(* PLC project AutomationML, AutomationML AutomationML AutomationML, author AutomationML *)
(* stored: creationDateTime 2017-02-14T12:09:57, companyURL AutomationML, productRelease AutomationML, language en-US, version AutomationML, organization AutomationML, modificationDateTime 2022-02-26T19:00:26 *)

PROGRAM Sequencing_Station_ActivityOnNodeNetwork
  VAR
    TA_030RB_300_takes_over_good : BOOL;
    TA_005RB_002_positions_workpiece1 : BOOL;
    TA_005RB_001_takes_over_workpiece1 : BOOL;
    TA_004CT_001_execute_trimming : BOOL;
    TA_003RB_002_positions_workpiece1 : BOOL;
    TA_001RB_001_takes_over_blank : BOOL;
    TA_001RB_002_positions_blank : BOOL;
    TA_030GST100_declamps_good : BOOL;
    TA_Execute_manufacturing_030RB_200 : BOOL;
    TA_Execute_manufacturing_030RB_100 : BOOL;
    TA_030GST100_clamps_goods : BOOL;
    TA_010RB_100_positions_workpiece1 : BOOL;
    TA_010RB_100_takes_over_workpiece1 : BOOL;
    TA_002DDP_001_execute_forming : BOOL;
    TA_003RB_001_takes_over_workpiece1 : BOOL;
    TA_006CMM_001_execute_cmm : BOOL;
    TA_007RB_001_takes_over_hinge_reinforcement : BOOL;
    TA_007RB_001_positions_hinge_reinforcement : BOOL;
    TA_030RB_300_positions_good : BOOL;
    TA_010UT_001_execute_inspection : BOOL;
  END_VAR

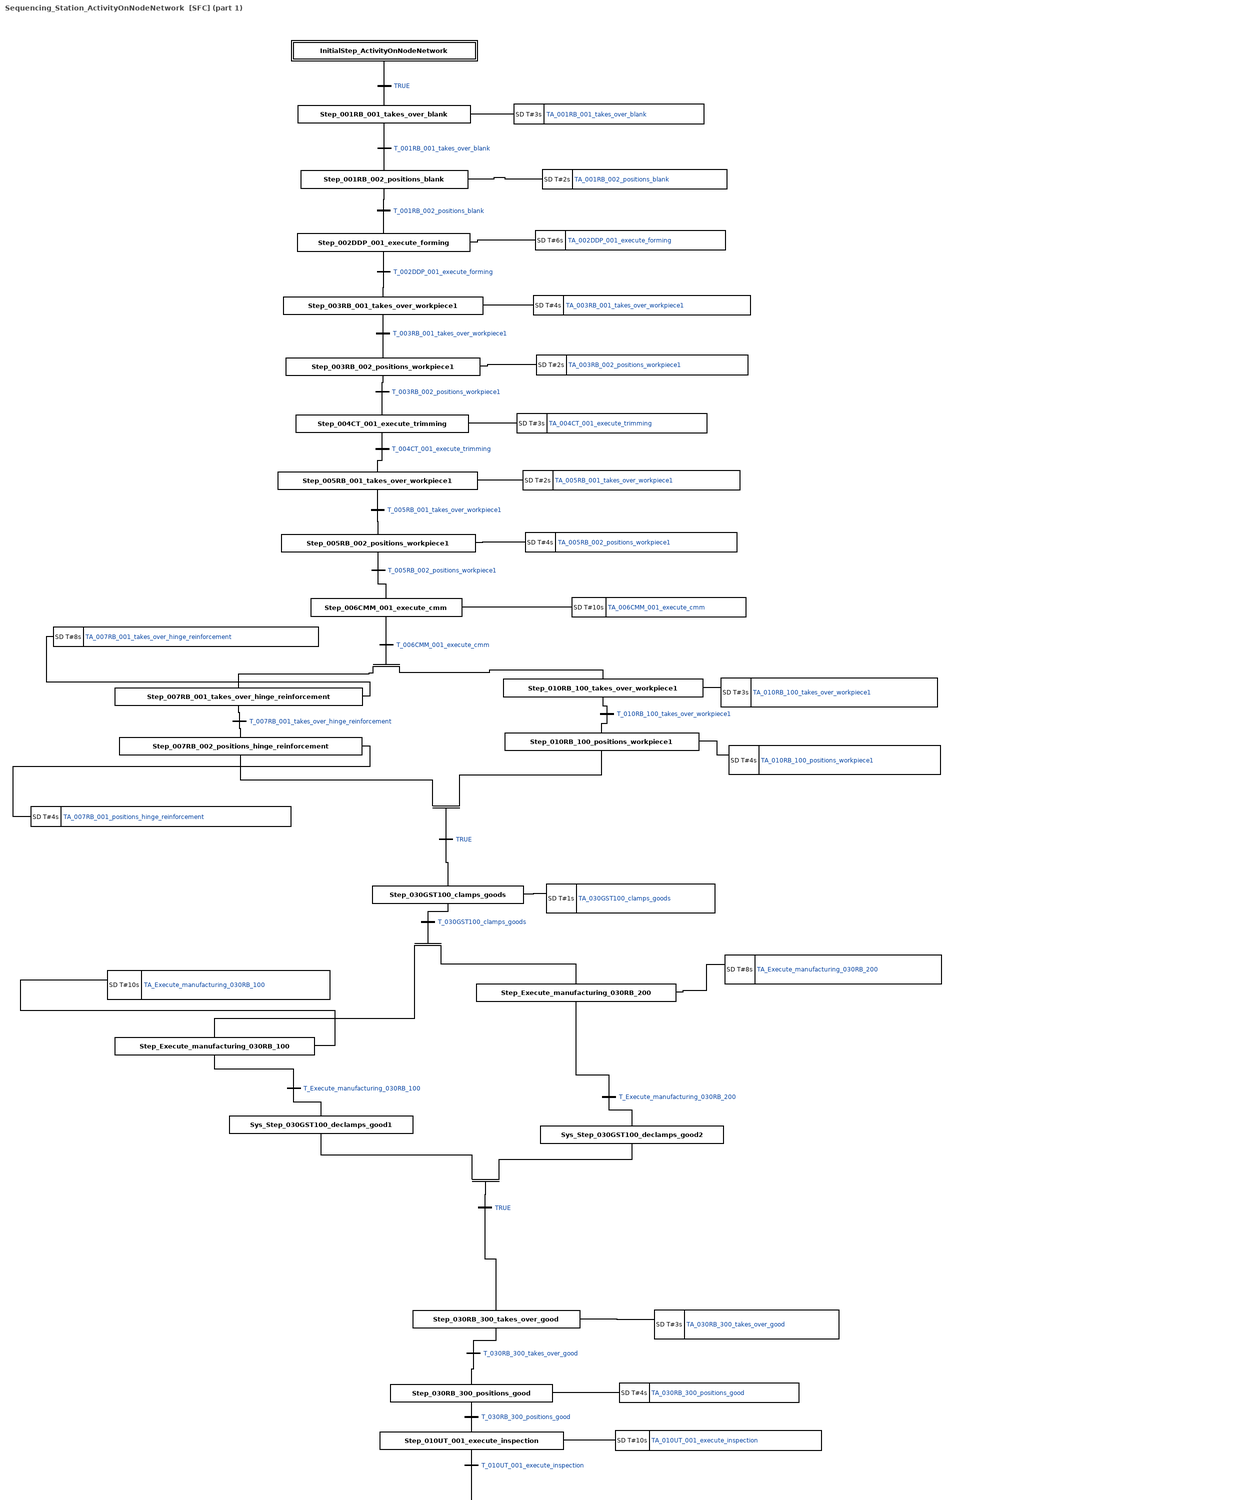
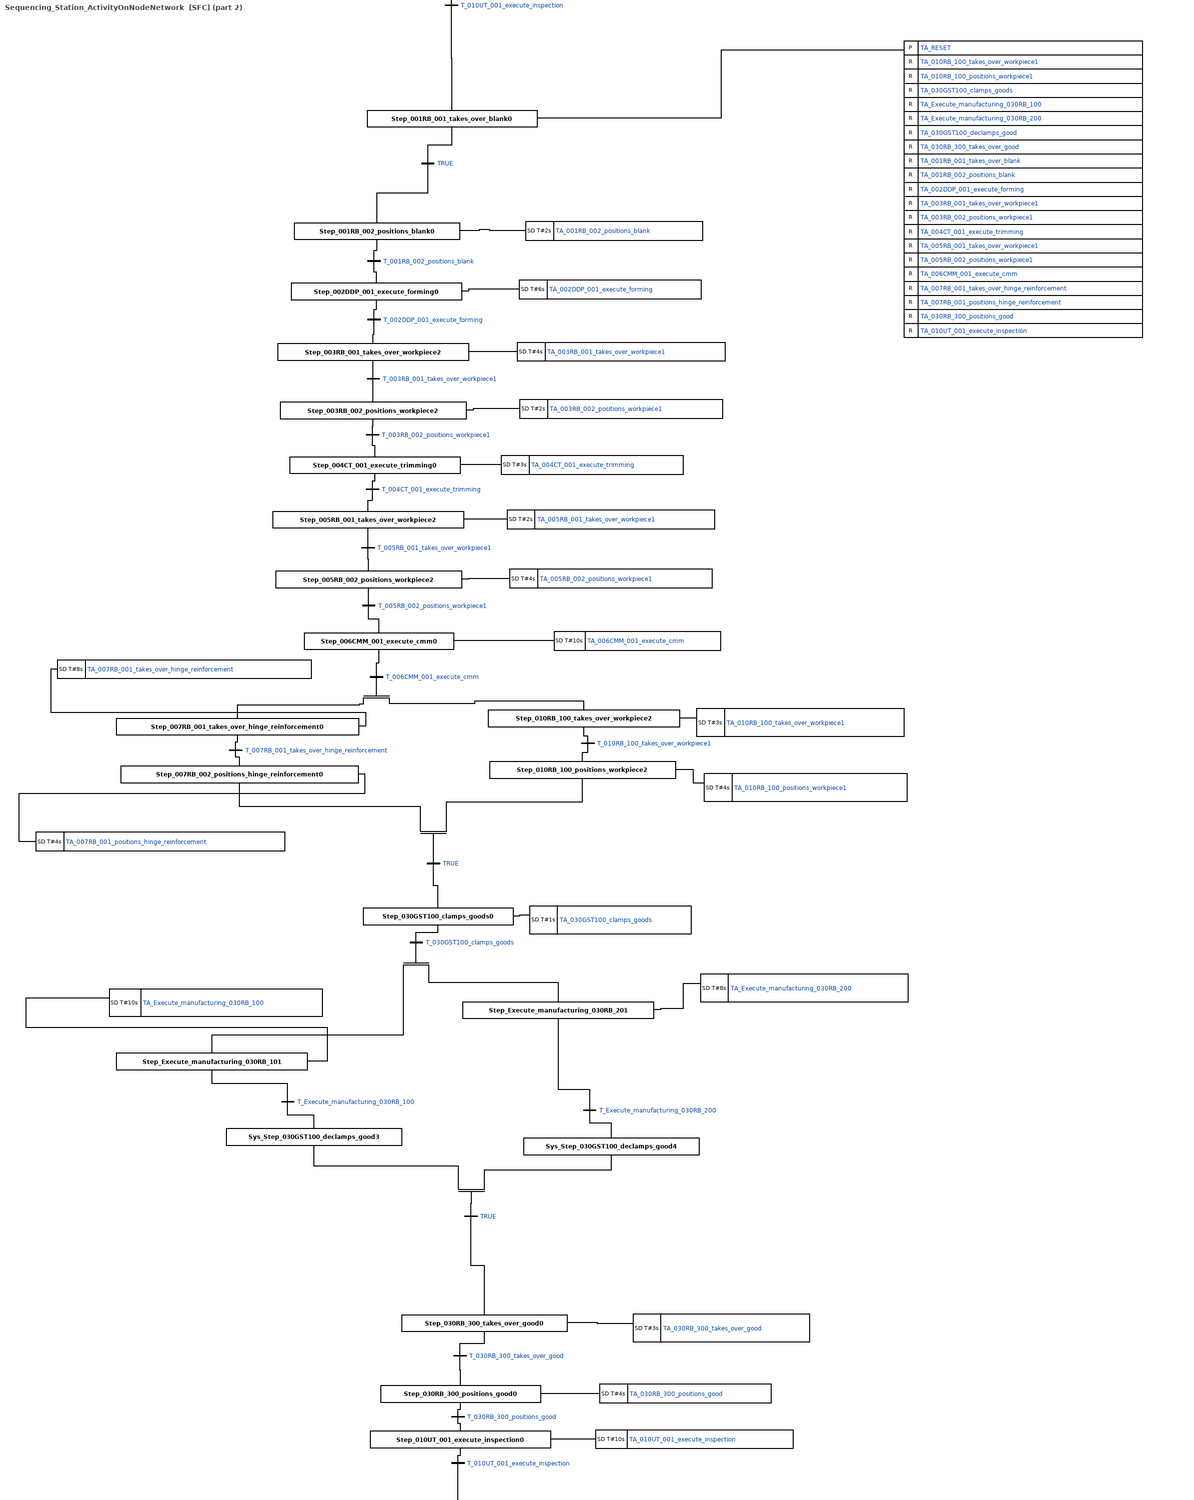
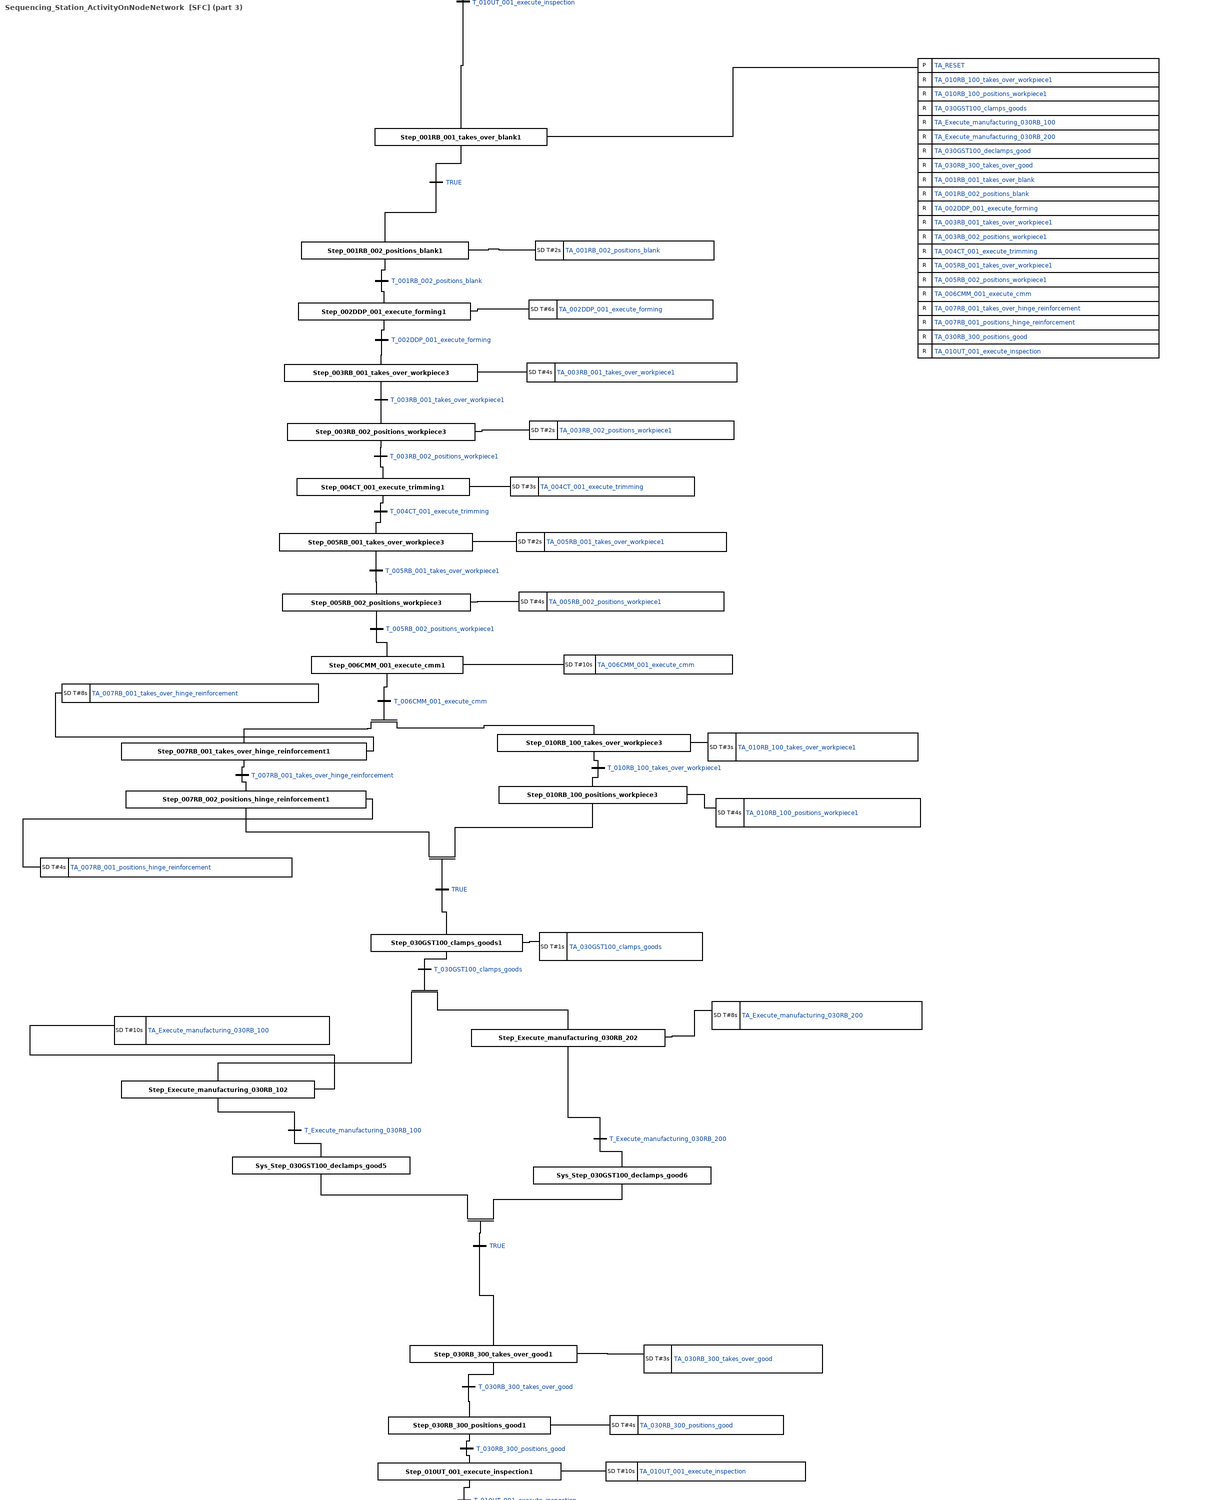
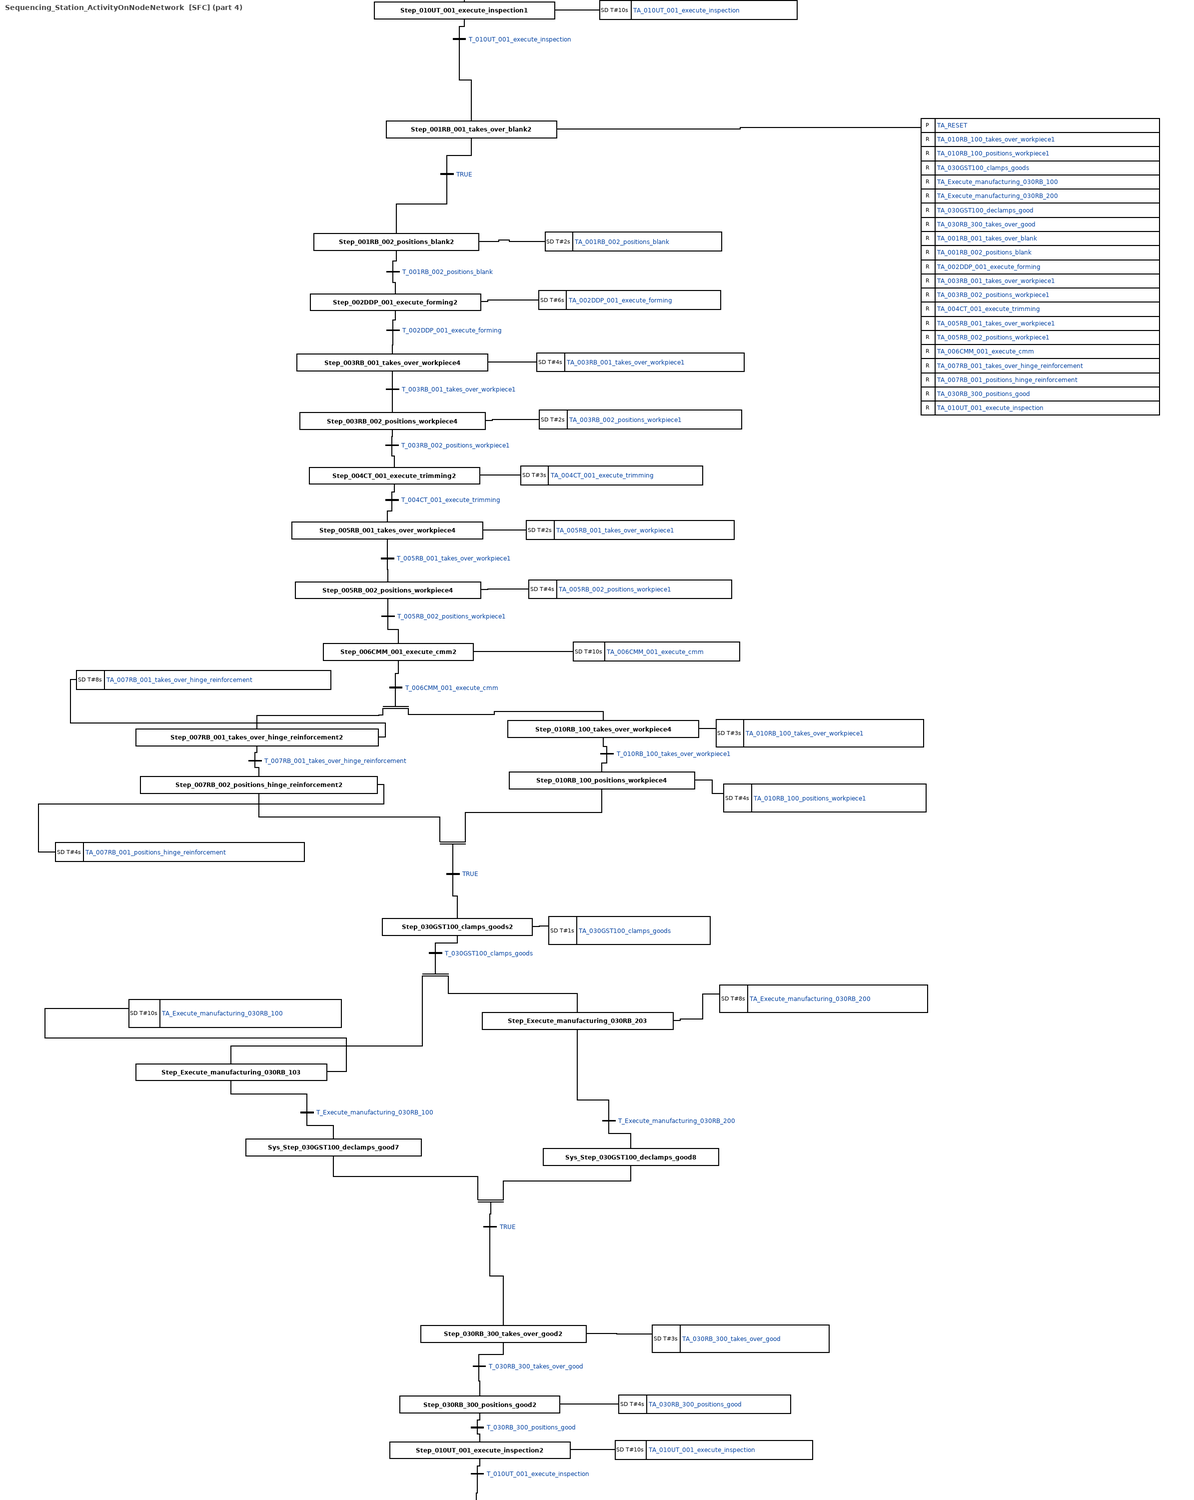
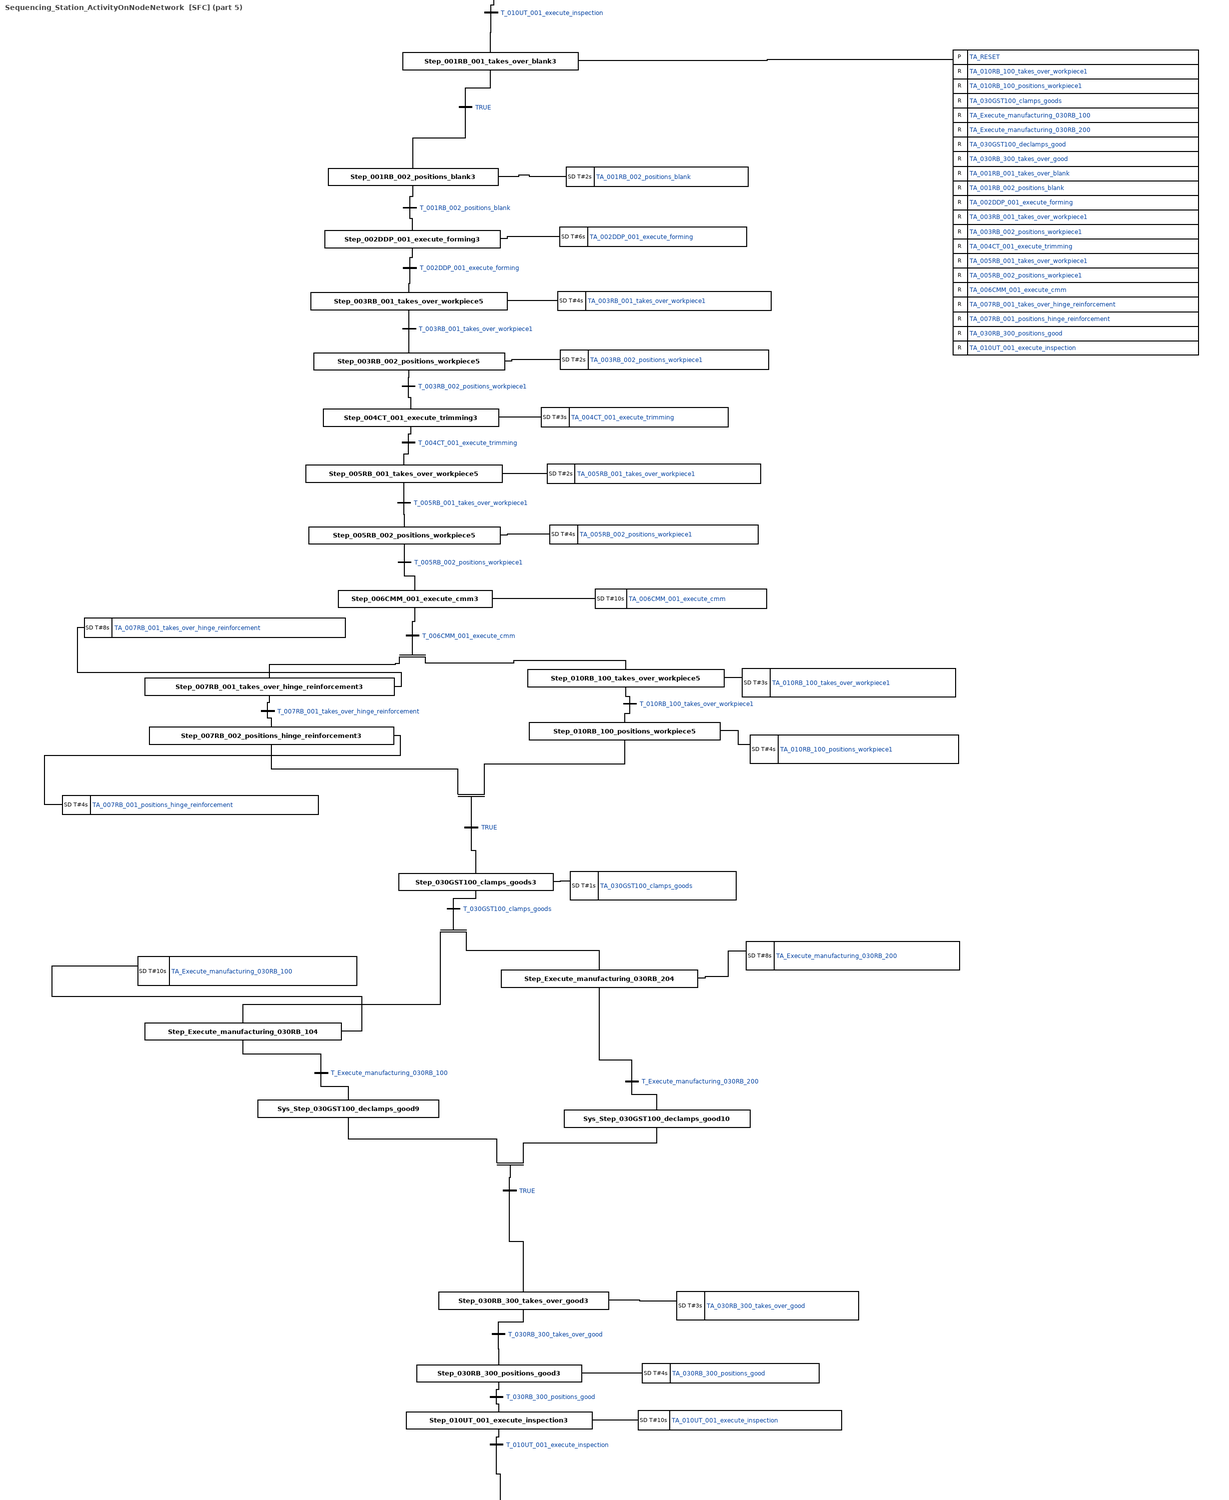
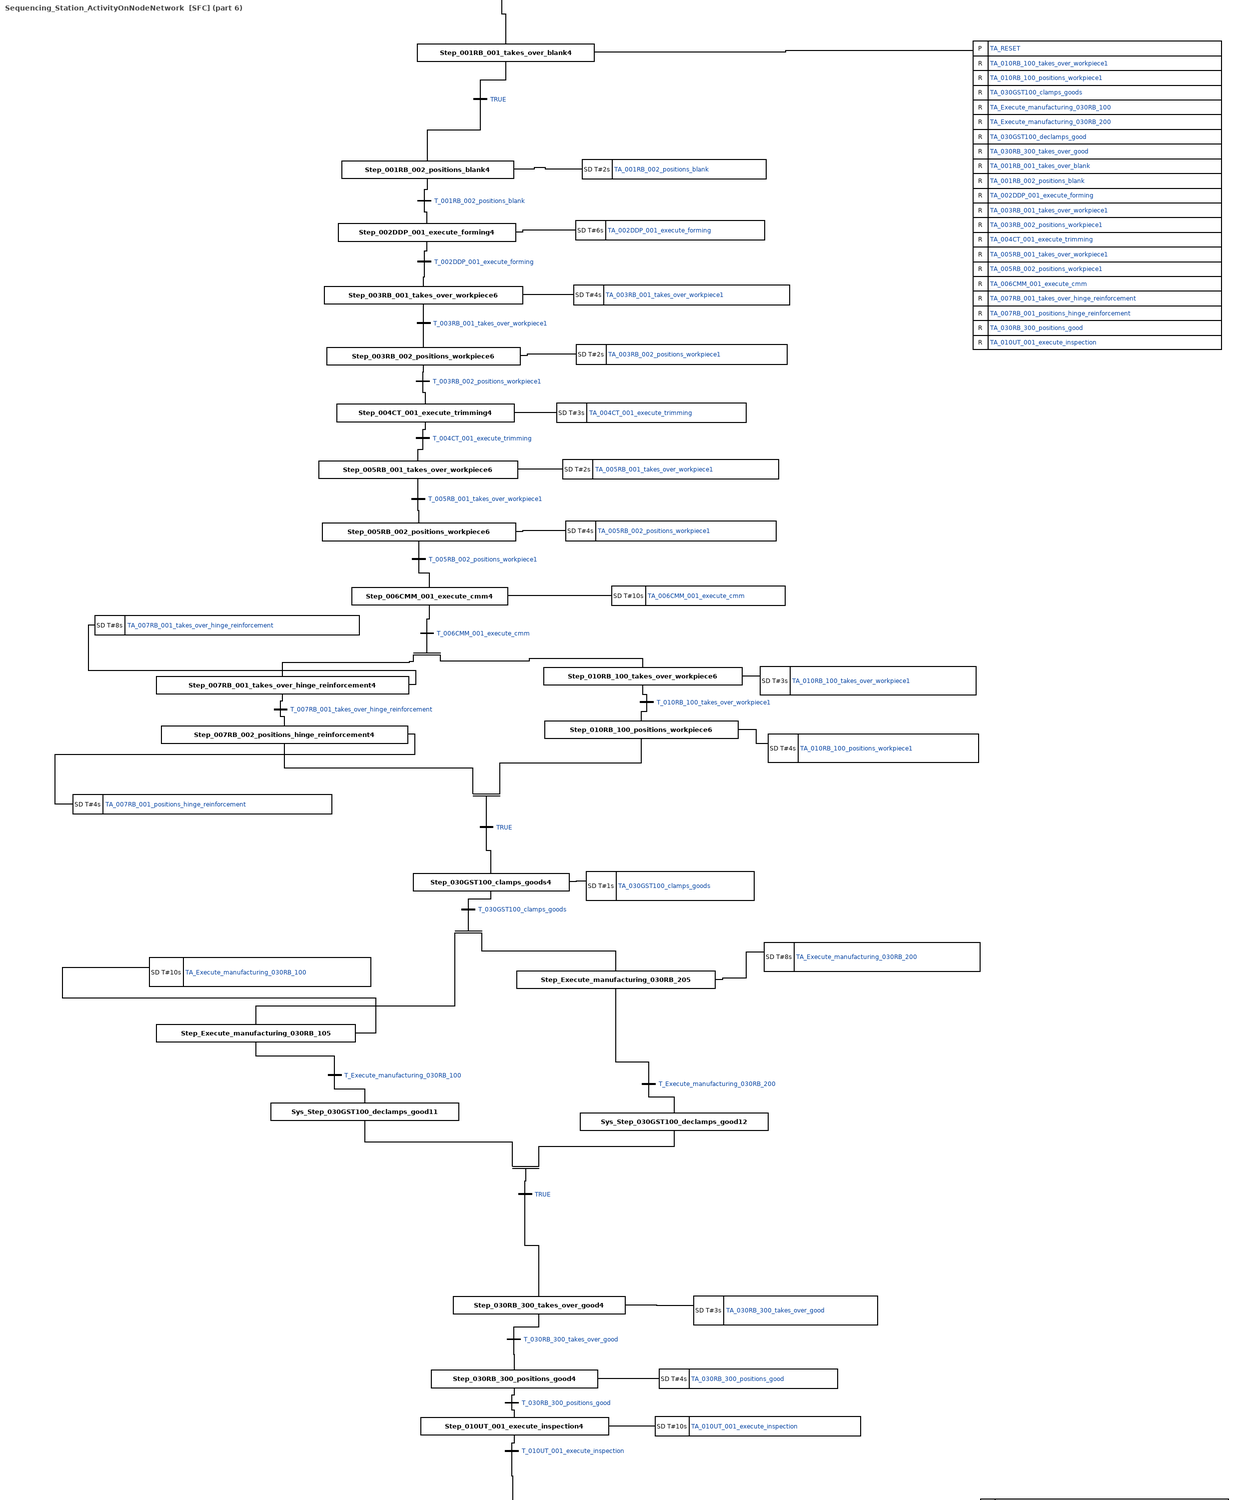
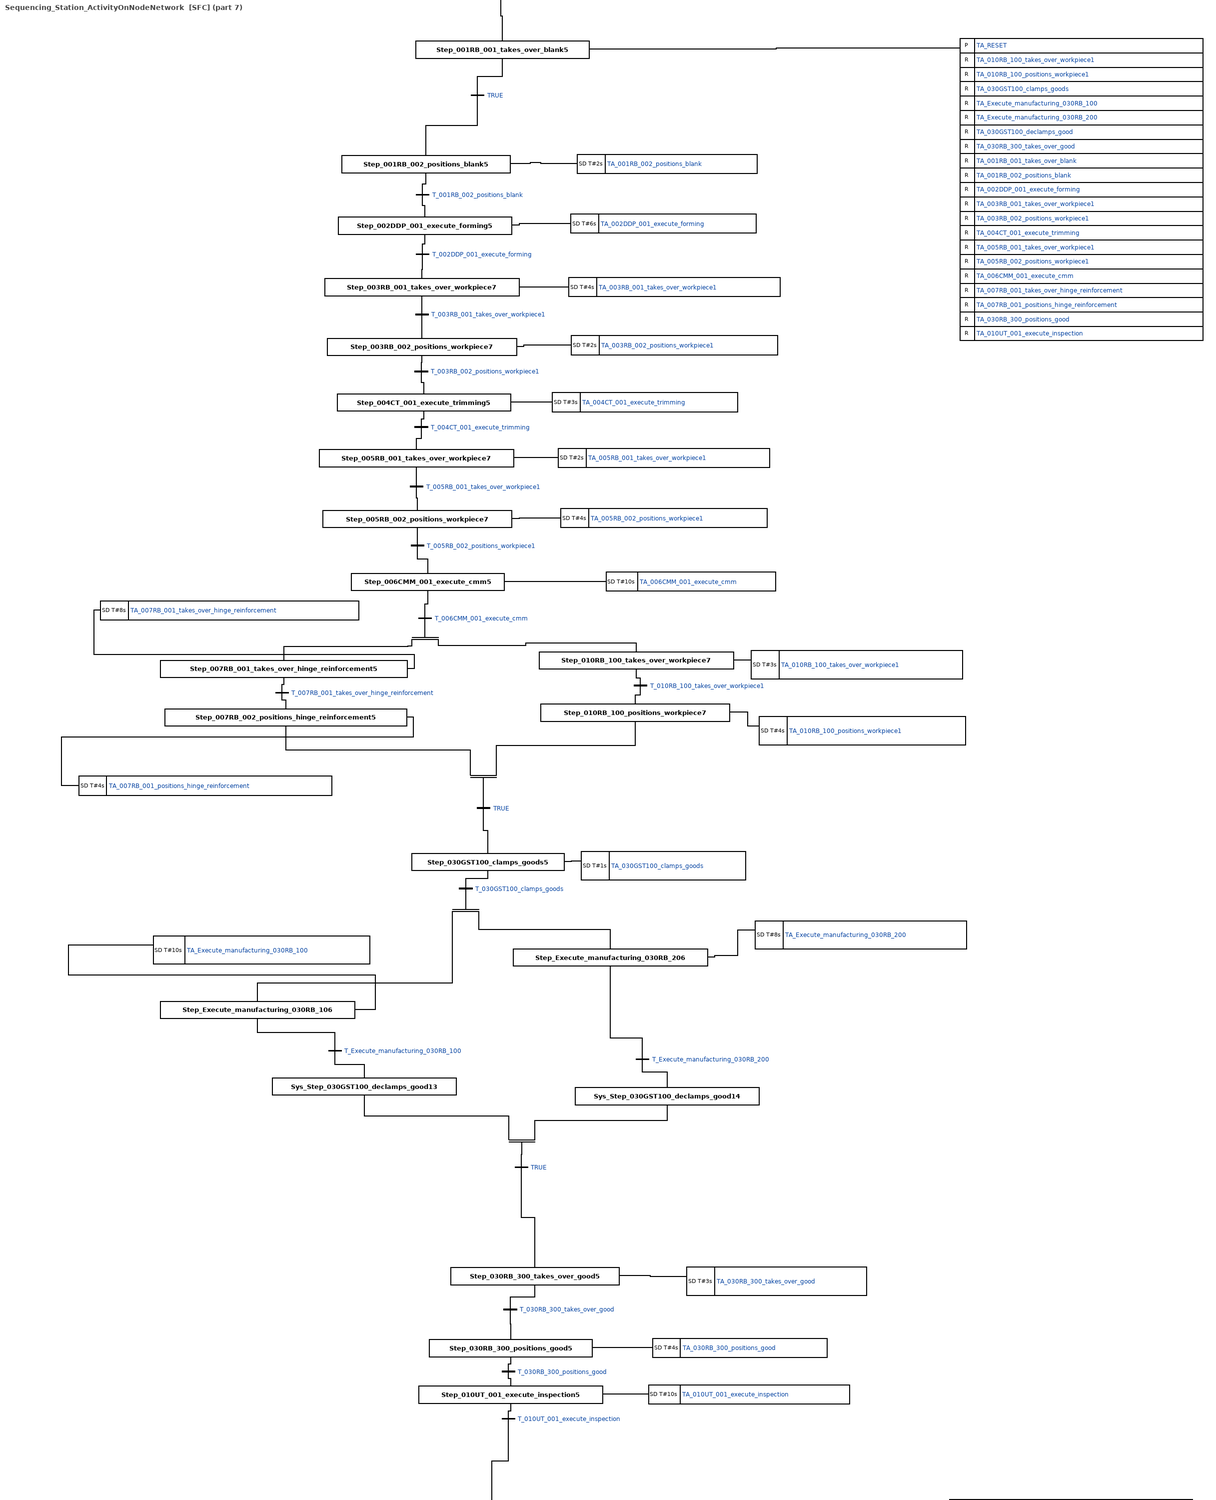
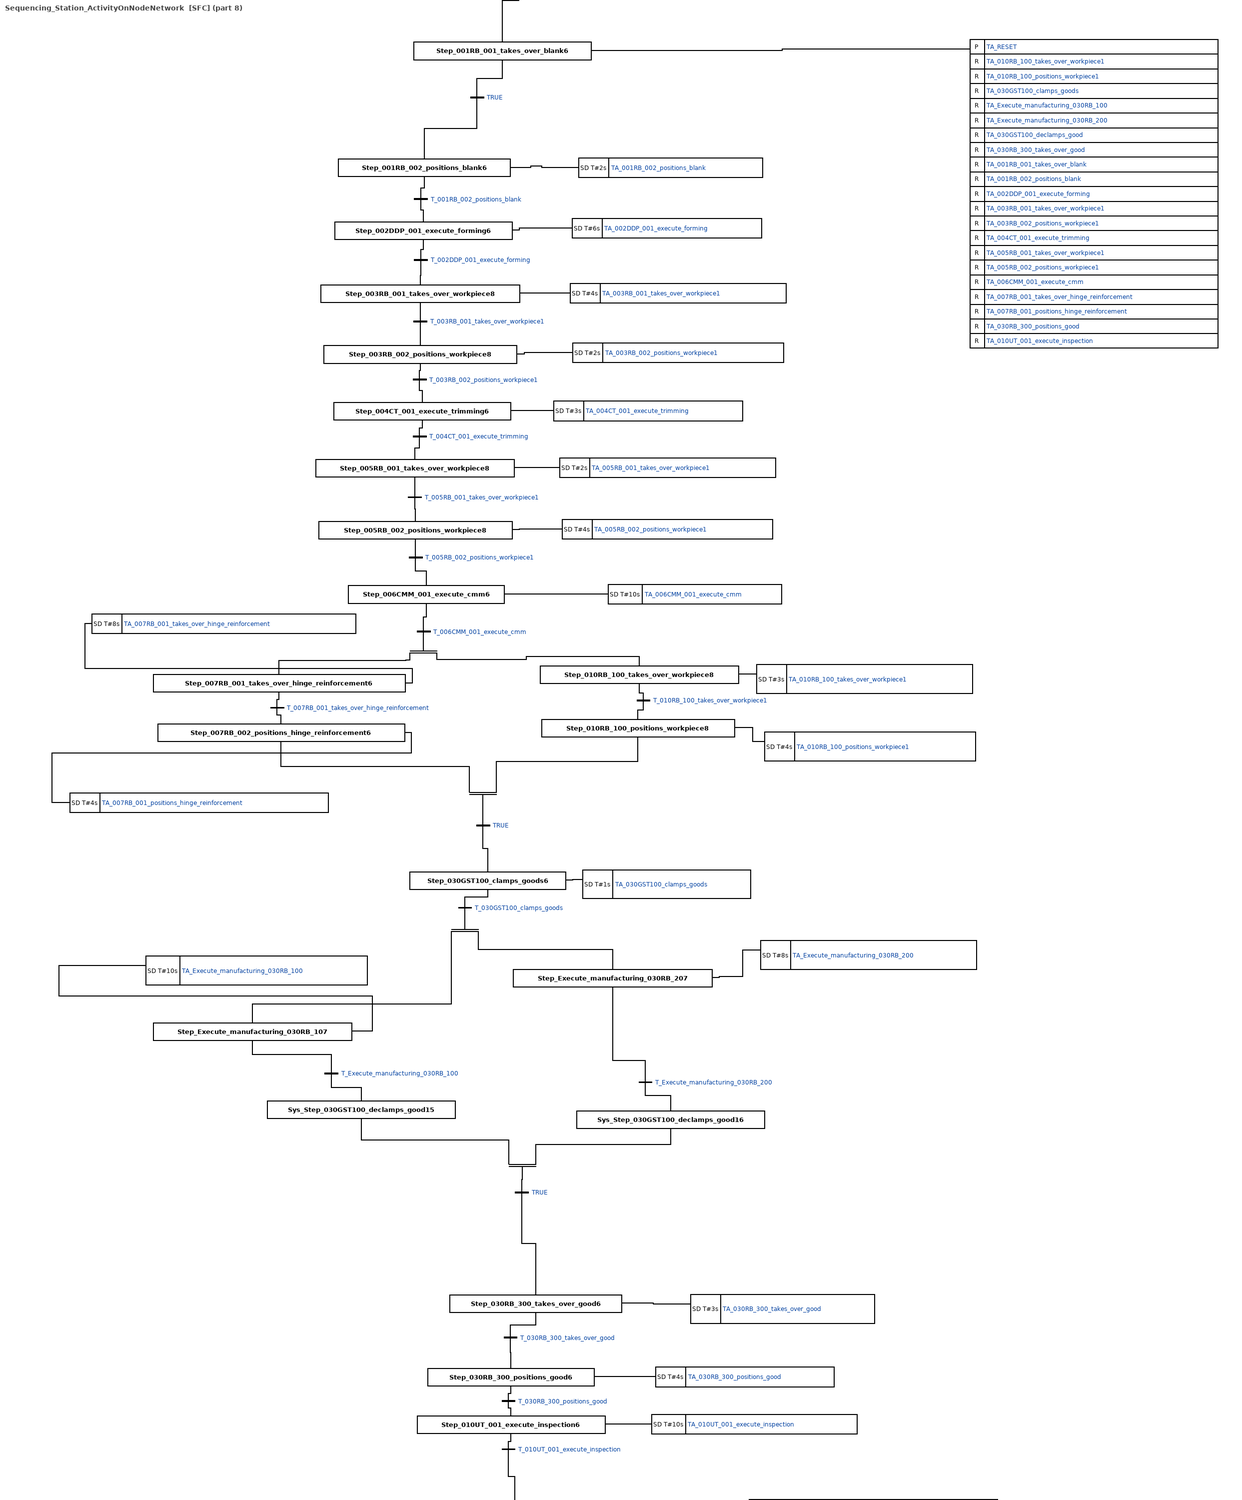
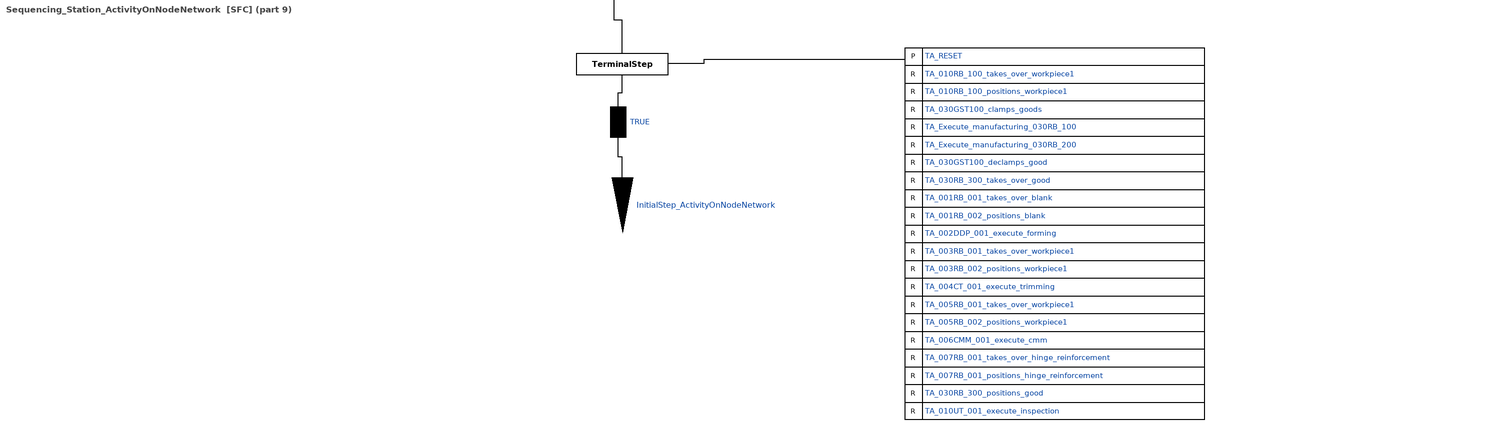
INITIAL_STEP InitialStep_ActivityOnNodeNetwork:
END_STEP
TRANSITION FROM InitialStep_ActivityOnNodeNetwork TO Step_001RB_001_takes_over_blank
  := TRUE;
END_TRANSITION
STEP Step_001RB_001_takes_over_blank:
  TA_001RB_001_takes_over_blank(SD, T#3s);
END_STEP
TRANSITION FROM Step_001RB_001_takes_over_blank TO Step_001RB_002_positions_blank  (* T_001RB_001_takes_over_blank *)
  := TA_001RB_001_takes_over_blank;
END_TRANSITION
STEP Step_001RB_002_positions_blank:
  TA_001RB_002_positions_blank(SD, T#2s);
END_STEP
TRANSITION FROM Step_001RB_002_positions_blank TO Step_002DDP_001_execute_forming  (* T_001RB_002_positions_blank *)
  := TA_001RB_002_positions_blank;
END_TRANSITION
STEP Step_002DDP_001_execute_forming:
  TA_002DDP_001_execute_forming(SD, T#6s);
END_STEP
TRANSITION FROM Step_002DDP_001_execute_forming TO Step_003RB_001_takes_over_workpiece1  (* T_002DDP_001_execute_forming *)
  := TA_002DDP_001_EXECUTE_FORMING;
END_TRANSITION
STEP Step_003RB_001_takes_over_workpiece1:
  TA_003RB_001_takes_over_workpiece1(SD, T#4s);
END_STEP
TRANSITION FROM Step_003RB_001_takes_over_workpiece1 TO Step_003RB_002_positions_workpiece1  (* T_003RB_001_takes_over_workpiece1 *)
  := TA_003RB_001_takes_over_workpiece1;
END_TRANSITION
STEP Step_003RB_002_positions_workpiece1:
  TA_003RB_002_positions_workpiece1(SD, T#2s);
END_STEP
TRANSITION FROM Step_003RB_002_positions_workpiece1 TO Step_004CT_001_execute_trimming  (* T_003RB_002_positions_workpiece1 *)
  := TA_003RB_002_positions_workpiece1;
END_TRANSITION
STEP Step_004CT_001_execute_trimming:
  TA_004CT_001_execute_trimming(SD, T#3s);
END_STEP
TRANSITION FROM Step_004CT_001_execute_trimming TO Step_005RB_001_takes_over_workpiece1  (* T_004CT_001_execute_trimming *)
  := TA_004CT_001_execute_trimming;
END_TRANSITION
STEP Step_005RB_001_takes_over_workpiece1:
  TA_005RB_001_takes_over_workpiece1(SD, T#2s);
END_STEP
TRANSITION FROM Step_005RB_001_takes_over_workpiece1 TO Step_005RB_002_positions_workpiece1  (* T_005RB_001_takes_over_workpiece1 *)
  := TA_005RB_001_takes_over_workpiece1;
END_TRANSITION
STEP Step_005RB_002_positions_workpiece1:
  TA_005RB_002_positions_workpiece1(SD, T#4s);
END_STEP
TRANSITION FROM Step_005RB_002_positions_workpiece1 TO Step_006CMM_001_execute_cmm  (* T_005RB_002_positions_workpiece1 *)
  := TA_005RB_002_positions_workpiece1;
END_TRANSITION
STEP Step_006CMM_001_execute_cmm:
  TA_006CMM_001_execute_cmm(SD, T#10s);
END_STEP
TRANSITION FROM Step_006CMM_001_execute_cmm TO (Step_010RB_100_takes_over_workpiece1, Step_007RB_001_takes_over_hinge_reinforcement)  (* T_006CMM_001_execute_cmm *)
  := TA_006CMM_001_execute_cmm;
END_TRANSITION
STEP Step_010RB_100_takes_over_workpiece1:
  TA_010RB_100_takes_over_workpiece1(SD, T#3s);
END_STEP
TRANSITION FROM Step_010RB_100_takes_over_workpiece1 TO Step_010RB_100_positions_workpiece1  (* T_010RB_100_takes_over_workpiece1 *)
  := TA_010RB_100_TAKES_OVER_WORKPIECE1;
END_TRANSITION
STEP Step_007RB_001_takes_over_hinge_reinforcement:
  TA_007RB_001_takes_over_hinge_reinforcement(SD, T#8s);
END_STEP
TRANSITION FROM Step_007RB_001_takes_over_hinge_reinforcement TO Step_007RB_002_positions_hinge_reinforcement  (* T_007RB_001_takes_over_hinge_reinforcement *)
  := TA_007RB_001_TAKES_OVER_HINGE_REINFORCEMENT;
END_TRANSITION
STEP Step_010RB_100_positions_workpiece1:
  TA_010RB_100_positions_workpiece1(SD, T#4s);
END_STEP
STEP Step_007RB_002_positions_hinge_reinforcement:
  TA_007RB_001_positions_hinge_reinforcement(SD, T#4s);
END_STEP
TRANSITION FROM (Step_007RB_002_positions_hinge_reinforcement, Step_010RB_100_positions_workpiece1) TO Step_030GST100_clamps_goods
  := TRUE;
END_TRANSITION
STEP Step_030GST100_clamps_goods:
  TA_030GST100_clamps_goods(SD, T#1s);
END_STEP
TRANSITION FROM Step_030GST100_clamps_goods TO (Step_Execute_manufacturing_030RB_100, Step_Execute_manufacturing_030RB_200)  (* T_030GST100_clamps_goods *)
  := TA_030GST100_clamps_goods;
END_TRANSITION
STEP Step_Execute_manufacturing_030RB_200:
  TA_Execute_manufacturing_030RB_200(SD, T#8s);
END_STEP
TRANSITION FROM Step_Execute_manufacturing_030RB_200 TO Sys_Step_030GST100_declamps_good2  (* T_Execute_manufacturing_030RB_200 *)
  := TA_Execute_manufacturing_030RB_200;
END_TRANSITION
STEP Step_Execute_manufacturing_030RB_100:
  TA_Execute_manufacturing_030RB_100(SD, T#10s);
END_STEP
TRANSITION FROM Step_Execute_manufacturing_030RB_100 TO Sys_Step_030GST100_declamps_good1  (* T_Execute_manufacturing_030RB_100 *)
  := TA_Execute_manufacturing_030RB_100;
END_TRANSITION
STEP Sys_Step_030GST100_declamps_good1:
END_STEP
TRANSITION FROM (Sys_Step_030GST100_declamps_good1, Sys_Step_030GST100_declamps_good2) TO Step_030RB_300_takes_over_good
  := TRUE;
END_TRANSITION
STEP Sys_Step_030GST100_declamps_good2:
END_STEP
STEP Step_030RB_300_takes_over_good:
  TA_030RB_300_takes_over_good(SD, T#3s);
END_STEP
TRANSITION FROM Step_030RB_300_takes_over_good TO Step_030RB_300_positions_good  (* T_030RB_300_takes_over_good *)
  := TA_030RB_300_takes_over_good;
END_TRANSITION
STEP Step_030RB_300_positions_good:
  TA_030RB_300_positions_good(SD, T#4s);
END_STEP
TRANSITION FROM Step_030RB_300_positions_good TO Step_010UT_001_execute_inspection  (* T_030RB_300_positions_good *)
  := TA_030RB_300_POSITIONS_GOOD;
END_TRANSITION
STEP Step_010UT_001_execute_inspection:
  TA_010UT_001_execute_inspection(SD, T#10s);
END_STEP
TRANSITION FROM Step_010UT_001_execute_inspection TO Step_001RB_001_takes_over_blank0  (* T_010UT_001_execute_inspection *)
  := TA_010UT_001_execute_inspection;
END_TRANSITION
STEP Step_001RB_001_takes_over_blank0:
  TA_RESET(P);
  TA_010RB_100_takes_over_workpiece1(R);
  TA_010RB_100_positions_workpiece1(R);
  TA_030GST100_clamps_goods(R);
  TA_Execute_manufacturing_030RB_100(R);
  TA_Execute_manufacturing_030RB_200(R);
  TA_030GST100_declamps_good(R);
  TA_030RB_300_takes_over_good(R);
  TA_001RB_001_takes_over_blank(R);
  TA_001RB_002_positions_blank(R);
  TA_002DDP_001_execute_forming(R);
  TA_003RB_001_takes_over_workpiece1(R);
  TA_003RB_002_positions_workpiece1(R);
  TA_004CT_001_execute_trimming(R);
  TA_005RB_001_takes_over_workpiece1(R);
  TA_005RB_002_positions_workpiece1(R);
  TA_006CMM_001_execute_cmm(R);
  TA_007RB_001_takes_over_hinge_reinforcement(R);
  TA_007RB_001_positions_hinge_reinforcement(R);
  TA_030RB_300_positions_good(R);
  TA_010UT_001_execute_inspection(R);
END_STEP
TRANSITION FROM Step_001RB_001_takes_over_blank0 TO Step_001RB_002_positions_blank0
  := TRUE;
END_TRANSITION
STEP Step_001RB_002_positions_blank0:
  TA_001RB_002_positions_blank(SD, T#2s);
END_STEP
TRANSITION FROM Step_001RB_002_positions_blank0 TO Step_002DDP_001_execute_forming0  (* T_001RB_002_positions_blank *)
  := TA_001RB_002_positions_blank;
END_TRANSITION
STEP Step_002DDP_001_execute_forming0:
  TA_002DDP_001_execute_forming(SD, T#6s);
END_STEP
TRANSITION FROM Step_002DDP_001_execute_forming0 TO Step_003RB_001_takes_over_workpiece2  (* T_002DDP_001_execute_forming *)
  := TA_002DDP_001_EXECUTE_FORMING;
END_TRANSITION
STEP Step_003RB_001_takes_over_workpiece2:
  TA_003RB_001_takes_over_workpiece1(SD, T#4s);
END_STEP
TRANSITION FROM Step_003RB_001_takes_over_workpiece2 TO Step_003RB_002_positions_workpiece2  (* T_003RB_001_takes_over_workpiece1 *)
  := TA_003RB_001_takes_over_workpiece1;
END_TRANSITION
STEP Step_003RB_002_positions_workpiece2:
  TA_003RB_002_positions_workpiece1(SD, T#2s);
END_STEP
TRANSITION FROM Step_003RB_002_positions_workpiece2 TO Step_004CT_001_execute_trimming0  (* T_003RB_002_positions_workpiece1 *)
  := TA_003RB_002_positions_workpiece1;
END_TRANSITION
STEP Step_004CT_001_execute_trimming0:
  TA_004CT_001_execute_trimming(SD, T#3s);
END_STEP
TRANSITION FROM Step_004CT_001_execute_trimming0 TO Step_005RB_001_takes_over_workpiece2  (* T_004CT_001_execute_trimming *)
  := TA_004CT_001_execute_trimming;
END_TRANSITION
STEP Step_005RB_001_takes_over_workpiece2:
  TA_005RB_001_takes_over_workpiece1(SD, T#2s);
END_STEP
TRANSITION FROM Step_005RB_001_takes_over_workpiece2 TO Step_005RB_002_positions_workpiece2  (* T_005RB_001_takes_over_workpiece1 *)
  := TA_005RB_001_takes_over_workpiece1;
END_TRANSITION
STEP Step_005RB_002_positions_workpiece2:
  TA_005RB_002_positions_workpiece1(SD, T#4s);
END_STEP
TRANSITION FROM Step_005RB_002_positions_workpiece2 TO Step_006CMM_001_execute_cmm0  (* T_005RB_002_positions_workpiece1 *)
  := TA_005RB_002_positions_workpiece1;
END_TRANSITION
STEP Step_006CMM_001_execute_cmm0:
  TA_006CMM_001_execute_cmm(SD, T#10s);
END_STEP
TRANSITION FROM Step_006CMM_001_execute_cmm0 TO (Step_010RB_100_takes_over_workpiece2, Step_007RB_001_takes_over_hinge_reinforcement0)  (* T_006CMM_001_execute_cmm *)
  := TA_006CMM_001_execute_cmm;
END_TRANSITION
STEP Step_010RB_100_takes_over_workpiece2:
  TA_010RB_100_takes_over_workpiece1(SD, T#3s);
END_STEP
TRANSITION FROM Step_010RB_100_takes_over_workpiece2 TO Step_010RB_100_positions_workpiece2  (* T_010RB_100_takes_over_workpiece1 *)
  := TA_010RB_100_TAKES_OVER_WORKPIECE1;
END_TRANSITION
STEP Step_007RB_001_takes_over_hinge_reinforcement0:
  TA_007RB_001_takes_over_hinge_reinforcement(SD, T#8s);
END_STEP
TRANSITION FROM Step_007RB_001_takes_over_hinge_reinforcement0 TO Step_007RB_002_positions_hinge_reinforcement0  (* T_007RB_001_takes_over_hinge_reinforcement *)
  := TA_007RB_001_TAKES_OVER_HINGE_REINFORCEMENT;
END_TRANSITION
STEP Step_010RB_100_positions_workpiece2:
  TA_010RB_100_positions_workpiece1(SD, T#4s);
END_STEP
STEP Step_007RB_002_positions_hinge_reinforcement0:
  TA_007RB_001_positions_hinge_reinforcement(SD, T#4s);
END_STEP
TRANSITION FROM (Step_007RB_002_positions_hinge_reinforcement0, Step_010RB_100_positions_workpiece2) TO Step_030GST100_clamps_goods0
  := TRUE;
END_TRANSITION
STEP Step_030GST100_clamps_goods0:
  TA_030GST100_clamps_goods(SD, T#1s);
END_STEP
TRANSITION FROM Step_030GST100_clamps_goods0 TO (Step_Execute_manufacturing_030RB_101, Step_Execute_manufacturing_030RB_201)  (* T_030GST100_clamps_goods *)
  := TA_030GST100_clamps_goods;
END_TRANSITION
STEP Step_Execute_manufacturing_030RB_201:
  TA_Execute_manufacturing_030RB_200(SD, T#8s);
END_STEP
TRANSITION FROM Step_Execute_manufacturing_030RB_201 TO Sys_Step_030GST100_declamps_good4  (* T_Execute_manufacturing_030RB_200 *)
  := TA_Execute_manufacturing_030RB_200;
END_TRANSITION
STEP Step_Execute_manufacturing_030RB_101:
  TA_Execute_manufacturing_030RB_100(SD, T#10s);
END_STEP
TRANSITION FROM Step_Execute_manufacturing_030RB_101 TO Sys_Step_030GST100_declamps_good3  (* T_Execute_manufacturing_030RB_100 *)
  := TA_Execute_manufacturing_030RB_100;
END_TRANSITION
STEP Sys_Step_030GST100_declamps_good3:
END_STEP
TRANSITION FROM (Sys_Step_030GST100_declamps_good3, Sys_Step_030GST100_declamps_good4) TO Step_030RB_300_takes_over_good0
  := TRUE;
END_TRANSITION
STEP Sys_Step_030GST100_declamps_good4:
END_STEP
STEP Step_030RB_300_takes_over_good0:
  TA_030RB_300_takes_over_good(SD, T#3s);
END_STEP
TRANSITION FROM Step_030RB_300_takes_over_good0 TO Step_030RB_300_positions_good0  (* T_030RB_300_takes_over_good *)
  := TA_030RB_300_takes_over_good;
END_TRANSITION
STEP Step_030RB_300_positions_good0:
  TA_030RB_300_positions_good(SD, T#4s);
END_STEP
TRANSITION FROM Step_030RB_300_positions_good0 TO Step_010UT_001_execute_inspection0  (* T_030RB_300_positions_good *)
  := TA_030RB_300_POSITIONS_GOOD;
END_TRANSITION
STEP Step_010UT_001_execute_inspection0:
  TA_010UT_001_execute_inspection(SD, T#10s);
END_STEP
TRANSITION FROM Step_010UT_001_execute_inspection0 TO Step_001RB_001_takes_over_blank1  (* T_010UT_001_execute_inspection *)
  := TA_010UT_001_execute_inspection;
END_TRANSITION
STEP Step_001RB_001_takes_over_blank1:
  TA_RESET(P);
  TA_010RB_100_takes_over_workpiece1(R);
  TA_010RB_100_positions_workpiece1(R);
  TA_030GST100_clamps_goods(R);
  TA_Execute_manufacturing_030RB_100(R);
  TA_Execute_manufacturing_030RB_200(R);
  TA_030GST100_declamps_good(R);
  TA_030RB_300_takes_over_good(R);
  TA_001RB_001_takes_over_blank(R);
  TA_001RB_002_positions_blank(R);
  TA_002DDP_001_execute_forming(R);
  TA_003RB_001_takes_over_workpiece1(R);
  TA_003RB_002_positions_workpiece1(R);
  TA_004CT_001_execute_trimming(R);
  TA_005RB_001_takes_over_workpiece1(R);
  TA_005RB_002_positions_workpiece1(R);
  TA_006CMM_001_execute_cmm(R);
  TA_007RB_001_takes_over_hinge_reinforcement(R);
  TA_007RB_001_positions_hinge_reinforcement(R);
  TA_030RB_300_positions_good(R);
  TA_010UT_001_execute_inspection(R);
END_STEP
TRANSITION FROM Step_001RB_001_takes_over_blank1 TO Step_001RB_002_positions_blank1
  := TRUE;
END_TRANSITION
STEP Step_001RB_002_positions_blank1:
  TA_001RB_002_positions_blank(SD, T#2s);
END_STEP
TRANSITION FROM Step_001RB_002_positions_blank1 TO Step_002DDP_001_execute_forming1  (* T_001RB_002_positions_blank *)
  := TA_001RB_002_positions_blank;
END_TRANSITION
STEP Step_002DDP_001_execute_forming1:
  TA_002DDP_001_execute_forming(SD, T#6s);
END_STEP
TRANSITION FROM Step_002DDP_001_execute_forming1 TO Step_003RB_001_takes_over_workpiece3  (* T_002DDP_001_execute_forming *)
  := TA_002DDP_001_EXECUTE_FORMING;
END_TRANSITION
STEP Step_003RB_001_takes_over_workpiece3:
  TA_003RB_001_takes_over_workpiece1(SD, T#4s);
END_STEP
TRANSITION FROM Step_003RB_001_takes_over_workpiece3 TO Step_003RB_002_positions_workpiece3  (* T_003RB_001_takes_over_workpiece1 *)
  := TA_003RB_001_takes_over_workpiece1;
END_TRANSITION
STEP Step_003RB_002_positions_workpiece3:
  TA_003RB_002_positions_workpiece1(SD, T#2s);
END_STEP
TRANSITION FROM Step_003RB_002_positions_workpiece3 TO Step_004CT_001_execute_trimming1  (* T_003RB_002_positions_workpiece1 *)
  := TA_003RB_002_positions_workpiece1;
END_TRANSITION
STEP Step_004CT_001_execute_trimming1:
  TA_004CT_001_execute_trimming(SD, T#3s);
END_STEP
TRANSITION FROM Step_004CT_001_execute_trimming1 TO Step_005RB_001_takes_over_workpiece3  (* T_004CT_001_execute_trimming *)
  := TA_004CT_001_execute_trimming;
END_TRANSITION
STEP Step_005RB_001_takes_over_workpiece3:
  TA_005RB_001_takes_over_workpiece1(SD, T#2s);
END_STEP
TRANSITION FROM Step_005RB_001_takes_over_workpiece3 TO Step_005RB_002_positions_workpiece3  (* T_005RB_001_takes_over_workpiece1 *)
  := TA_005RB_001_takes_over_workpiece1;
END_TRANSITION
STEP Step_005RB_002_positions_workpiece3:
  TA_005RB_002_positions_workpiece1(SD, T#4s);
END_STEP
TRANSITION FROM Step_005RB_002_positions_workpiece3 TO Step_006CMM_001_execute_cmm1  (* T_005RB_002_positions_workpiece1 *)
  := TA_005RB_002_positions_workpiece1;
END_TRANSITION
STEP Step_006CMM_001_execute_cmm1:
  TA_006CMM_001_execute_cmm(SD, T#10s);
END_STEP
TRANSITION FROM Step_006CMM_001_execute_cmm1 TO (Step_010RB_100_takes_over_workpiece3, Step_007RB_001_takes_over_hinge_reinforcement1)  (* T_006CMM_001_execute_cmm *)
  := TA_006CMM_001_execute_cmm;
END_TRANSITION
STEP Step_010RB_100_takes_over_workpiece3:
  TA_010RB_100_takes_over_workpiece1(SD, T#3s);
END_STEP
TRANSITION FROM Step_010RB_100_takes_over_workpiece3 TO Step_010RB_100_positions_workpiece3  (* T_010RB_100_takes_over_workpiece1 *)
  := TA_010RB_100_TAKES_OVER_WORKPIECE1;
END_TRANSITION
STEP Step_007RB_001_takes_over_hinge_reinforcement1:
  TA_007RB_001_takes_over_hinge_reinforcement(SD, T#8s);
END_STEP
TRANSITION FROM Step_007RB_001_takes_over_hinge_reinforcement1 TO Step_007RB_002_positions_hinge_reinforcement1  (* T_007RB_001_takes_over_hinge_reinforcement *)
  := TA_007RB_001_TAKES_OVER_HINGE_REINFORCEMENT;
END_TRANSITION
STEP Step_010RB_100_positions_workpiece3:
  TA_010RB_100_positions_workpiece1(SD, T#4s);
END_STEP
STEP Step_007RB_002_positions_hinge_reinforcement1:
  TA_007RB_001_positions_hinge_reinforcement(SD, T#4s);
END_STEP
TRANSITION FROM (Step_007RB_002_positions_hinge_reinforcement1, Step_010RB_100_positions_workpiece3) TO Step_030GST100_clamps_goods1
  := TRUE;
END_TRANSITION
STEP Step_030GST100_clamps_goods1:
  TA_030GST100_clamps_goods(SD, T#1s);
END_STEP
TRANSITION FROM Step_030GST100_clamps_goods1 TO (Step_Execute_manufacturing_030RB_102, Step_Execute_manufacturing_030RB_202)  (* T_030GST100_clamps_goods *)
  := TA_030GST100_clamps_goods;
END_TRANSITION
STEP Step_Execute_manufacturing_030RB_202:
  TA_Execute_manufacturing_030RB_200(SD, T#8s);
END_STEP
TRANSITION FROM Step_Execute_manufacturing_030RB_202 TO Sys_Step_030GST100_declamps_good6  (* T_Execute_manufacturing_030RB_200 *)
  := TA_Execute_manufacturing_030RB_200;
END_TRANSITION
STEP Step_Execute_manufacturing_030RB_102:
  TA_Execute_manufacturing_030RB_100(SD, T#10s);
END_STEP
TRANSITION FROM Step_Execute_manufacturing_030RB_102 TO Sys_Step_030GST100_declamps_good5  (* T_Execute_manufacturing_030RB_100 *)
  := TA_Execute_manufacturing_030RB_100;
END_TRANSITION
STEP Sys_Step_030GST100_declamps_good5:
END_STEP
TRANSITION FROM (Sys_Step_030GST100_declamps_good5, Sys_Step_030GST100_declamps_good6) TO Step_030RB_300_takes_over_good1
  := TRUE;
END_TRANSITION
STEP Sys_Step_030GST100_declamps_good6:
END_STEP
STEP Step_030RB_300_takes_over_good1:
  TA_030RB_300_takes_over_good(SD, T#3s);
END_STEP
TRANSITION FROM Step_030RB_300_takes_over_good1 TO Step_030RB_300_positions_good1  (* T_030RB_300_takes_over_good *)
  := TA_030RB_300_takes_over_good;
END_TRANSITION
STEP Step_030RB_300_positions_good1:
  TA_030RB_300_positions_good(SD, T#4s);
END_STEP
TRANSITION FROM Step_030RB_300_positions_good1 TO Step_010UT_001_execute_inspection1  (* T_030RB_300_positions_good *)
  := TA_030RB_300_POSITIONS_GOOD;
END_TRANSITION
STEP Step_010UT_001_execute_inspection1:
  TA_010UT_001_execute_inspection(SD, T#10s);
END_STEP
TRANSITION FROM Step_010UT_001_execute_inspection1 TO Step_001RB_001_takes_over_blank2  (* T_010UT_001_execute_inspection *)
  := TA_010UT_001_execute_inspection;
END_TRANSITION
STEP Step_001RB_001_takes_over_blank2:
  TA_RESET(P);
  TA_010RB_100_takes_over_workpiece1(R);
  TA_010RB_100_positions_workpiece1(R);
  TA_030GST100_clamps_goods(R);
  TA_Execute_manufacturing_030RB_100(R);
  TA_Execute_manufacturing_030RB_200(R);
  TA_030GST100_declamps_good(R);
  TA_030RB_300_takes_over_good(R);
  TA_001RB_001_takes_over_blank(R);
  TA_001RB_002_positions_blank(R);
  TA_002DDP_001_execute_forming(R);
  TA_003RB_001_takes_over_workpiece1(R);
  TA_003RB_002_positions_workpiece1(R);
  TA_004CT_001_execute_trimming(R);
  TA_005RB_001_takes_over_workpiece1(R);
  TA_005RB_002_positions_workpiece1(R);
  TA_006CMM_001_execute_cmm(R);
  TA_007RB_001_takes_over_hinge_reinforcement(R);
  TA_007RB_001_positions_hinge_reinforcement(R);
  TA_030RB_300_positions_good(R);
  TA_010UT_001_execute_inspection(R);
END_STEP
TRANSITION FROM Step_001RB_001_takes_over_blank2 TO Step_001RB_002_positions_blank2
  := TRUE;
END_TRANSITION
STEP Step_001RB_002_positions_blank2:
  TA_001RB_002_positions_blank(SD, T#2s);
END_STEP
TRANSITION FROM Step_001RB_002_positions_blank2 TO Step_002DDP_001_execute_forming2  (* T_001RB_002_positions_blank *)
  := TA_001RB_002_positions_blank;
END_TRANSITION
STEP Step_002DDP_001_execute_forming2:
  TA_002DDP_001_execute_forming(SD, T#6s);
END_STEP
TRANSITION FROM Step_002DDP_001_execute_forming2 TO Step_003RB_001_takes_over_workpiece4  (* T_002DDP_001_execute_forming *)
  := TA_002DDP_001_EXECUTE_FORMING;
END_TRANSITION
STEP Step_003RB_001_takes_over_workpiece4:
  TA_003RB_001_takes_over_workpiece1(SD, T#4s);
END_STEP
TRANSITION FROM Step_003RB_001_takes_over_workpiece4 TO Step_003RB_002_positions_workpiece4  (* T_003RB_001_takes_over_workpiece1 *)
  := TA_003RB_001_takes_over_workpiece1;
END_TRANSITION
STEP Step_003RB_002_positions_workpiece4:
  TA_003RB_002_positions_workpiece1(SD, T#2s);
END_STEP
TRANSITION FROM Step_003RB_002_positions_workpiece4 TO Step_004CT_001_execute_trimming2  (* T_003RB_002_positions_workpiece1 *)
  := TA_003RB_002_positions_workpiece1;
END_TRANSITION
STEP Step_004CT_001_execute_trimming2:
  TA_004CT_001_execute_trimming(SD, T#3s);
END_STEP
TRANSITION FROM Step_004CT_001_execute_trimming2 TO Step_005RB_001_takes_over_workpiece4  (* T_004CT_001_execute_trimming *)
  := TA_004CT_001_execute_trimming;
END_TRANSITION
STEP Step_005RB_001_takes_over_workpiece4:
  TA_005RB_001_takes_over_workpiece1(SD, T#2s);
END_STEP
TRANSITION FROM Step_005RB_001_takes_over_workpiece4 TO Step_005RB_002_positions_workpiece4  (* T_005RB_001_takes_over_workpiece1 *)
  := TA_005RB_001_takes_over_workpiece1;
END_TRANSITION
STEP Step_005RB_002_positions_workpiece4:
  TA_005RB_002_positions_workpiece1(SD, T#4s);
END_STEP
TRANSITION FROM Step_005RB_002_positions_workpiece4 TO Step_006CMM_001_execute_cmm2  (* T_005RB_002_positions_workpiece1 *)
  := TA_005RB_002_positions_workpiece1;
END_TRANSITION
STEP Step_006CMM_001_execute_cmm2:
  TA_006CMM_001_execute_cmm(SD, T#10s);
END_STEP
TRANSITION FROM Step_006CMM_001_execute_cmm2 TO (Step_010RB_100_takes_over_workpiece4, Step_007RB_001_takes_over_hinge_reinforcement2)  (* T_006CMM_001_execute_cmm *)
  := TA_006CMM_001_execute_cmm;
END_TRANSITION
STEP Step_010RB_100_takes_over_workpiece4:
  TA_010RB_100_takes_over_workpiece1(SD, T#3s);
END_STEP
TRANSITION FROM Step_010RB_100_takes_over_workpiece4 TO Step_010RB_100_positions_workpiece4  (* T_010RB_100_takes_over_workpiece1 *)
  := TA_010RB_100_TAKES_OVER_WORKPIECE1;
END_TRANSITION
STEP Step_007RB_001_takes_over_hinge_reinforcement2:
  TA_007RB_001_takes_over_hinge_reinforcement(SD, T#8s);
END_STEP
TRANSITION FROM Step_007RB_001_takes_over_hinge_reinforcement2 TO Step_007RB_002_positions_hinge_reinforcement2  (* T_007RB_001_takes_over_hinge_reinforcement *)
  := TA_007RB_001_TAKES_OVER_HINGE_REINFORCEMENT;
END_TRANSITION
STEP Step_010RB_100_positions_workpiece4:
  TA_010RB_100_positions_workpiece1(SD, T#4s);
END_STEP
STEP Step_007RB_002_positions_hinge_reinforcement2:
  TA_007RB_001_positions_hinge_reinforcement(SD, T#4s);
END_STEP
TRANSITION FROM (Step_007RB_002_positions_hinge_reinforcement2, Step_010RB_100_positions_workpiece4) TO Step_030GST100_clamps_goods2
  := TRUE;
END_TRANSITION
STEP Step_030GST100_clamps_goods2:
  TA_030GST100_clamps_goods(SD, T#1s);
END_STEP
TRANSITION FROM Step_030GST100_clamps_goods2 TO (Step_Execute_manufacturing_030RB_103, Step_Execute_manufacturing_030RB_203)  (* T_030GST100_clamps_goods *)
  := TA_030GST100_clamps_goods;
END_TRANSITION
STEP Step_Execute_manufacturing_030RB_203:
  TA_Execute_manufacturing_030RB_200(SD, T#8s);
END_STEP
TRANSITION FROM Step_Execute_manufacturing_030RB_203 TO Sys_Step_030GST100_declamps_good8  (* T_Execute_manufacturing_030RB_200 *)
  := TA_Execute_manufacturing_030RB_200;
END_TRANSITION
STEP Step_Execute_manufacturing_030RB_103:
  TA_Execute_manufacturing_030RB_100(SD, T#10s);
END_STEP
TRANSITION FROM Step_Execute_manufacturing_030RB_103 TO Sys_Step_030GST100_declamps_good7  (* T_Execute_manufacturing_030RB_100 *)
  := TA_Execute_manufacturing_030RB_100;
END_TRANSITION
STEP Sys_Step_030GST100_declamps_good7:
END_STEP
TRANSITION FROM (Sys_Step_030GST100_declamps_good7, Sys_Step_030GST100_declamps_good8) TO Step_030RB_300_takes_over_good2
  := TRUE;
END_TRANSITION
STEP Sys_Step_030GST100_declamps_good8:
END_STEP
STEP Step_030RB_300_takes_over_good2:
  TA_030RB_300_takes_over_good(SD, T#3s);
END_STEP
TRANSITION FROM Step_030RB_300_takes_over_good2 TO Step_030RB_300_positions_good2  (* T_030RB_300_takes_over_good *)
  := TA_030RB_300_takes_over_good;
END_TRANSITION
STEP Step_030RB_300_positions_good2:
  TA_030RB_300_positions_good(SD, T#4s);
END_STEP
TRANSITION FROM Step_030RB_300_positions_good2 TO Step_010UT_001_execute_inspection2  (* T_030RB_300_positions_good *)
  := TA_030RB_300_POSITIONS_GOOD;
END_TRANSITION
STEP Step_010UT_001_execute_inspection2:
  TA_010UT_001_execute_inspection(SD, T#10s);
END_STEP
TRANSITION FROM Step_010UT_001_execute_inspection2 TO Step_001RB_001_takes_over_blank3  (* T_010UT_001_execute_inspection *)
  := TA_010UT_001_execute_inspection;
END_TRANSITION
STEP Step_001RB_001_takes_over_blank3:
  TA_RESET(P);
  TA_010RB_100_takes_over_workpiece1(R);
  TA_010RB_100_positions_workpiece1(R);
  TA_030GST100_clamps_goods(R);
  TA_Execute_manufacturing_030RB_100(R);
  TA_Execute_manufacturing_030RB_200(R);
  TA_030GST100_declamps_good(R);
  TA_030RB_300_takes_over_good(R);
  TA_001RB_001_takes_over_blank(R);
  TA_001RB_002_positions_blank(R);
  TA_002DDP_001_execute_forming(R);
  TA_003RB_001_takes_over_workpiece1(R);
  TA_003RB_002_positions_workpiece1(R);
  TA_004CT_001_execute_trimming(R);
  TA_005RB_001_takes_over_workpiece1(R);
  TA_005RB_002_positions_workpiece1(R);
  TA_006CMM_001_execute_cmm(R);
  TA_007RB_001_takes_over_hinge_reinforcement(R);
  TA_007RB_001_positions_hinge_reinforcement(R);
  TA_030RB_300_positions_good(R);
  TA_010UT_001_execute_inspection(R);
END_STEP
TRANSITION FROM Step_001RB_001_takes_over_blank3 TO Step_001RB_002_positions_blank3
  := TRUE;
END_TRANSITION
STEP Step_001RB_002_positions_blank3:
  TA_001RB_002_positions_blank(SD, T#2s);
END_STEP
TRANSITION FROM Step_001RB_002_positions_blank3 TO Step_002DDP_001_execute_forming3  (* T_001RB_002_positions_blank *)
  := TA_001RB_002_positions_blank;
END_TRANSITION
STEP Step_002DDP_001_execute_forming3:
  TA_002DDP_001_execute_forming(SD, T#6s);
END_STEP
TRANSITION FROM Step_002DDP_001_execute_forming3 TO Step_003RB_001_takes_over_workpiece5  (* T_002DDP_001_execute_forming *)
  := TA_002DDP_001_EXECUTE_FORMING;
END_TRANSITION
STEP Step_003RB_001_takes_over_workpiece5:
  TA_003RB_001_takes_over_workpiece1(SD, T#4s);
END_STEP
TRANSITION FROM Step_003RB_001_takes_over_workpiece5 TO Step_003RB_002_positions_workpiece5  (* T_003RB_001_takes_over_workpiece1 *)
  := TA_003RB_001_takes_over_workpiece1;
END_TRANSITION
STEP Step_003RB_002_positions_workpiece5:
  TA_003RB_002_positions_workpiece1(SD, T#2s);
END_STEP
TRANSITION FROM Step_003RB_002_positions_workpiece5 TO Step_004CT_001_execute_trimming3  (* T_003RB_002_positions_workpiece1 *)
  := TA_003RB_002_positions_workpiece1;
END_TRANSITION
STEP Step_004CT_001_execute_trimming3:
  TA_004CT_001_execute_trimming(SD, T#3s);
END_STEP
TRANSITION FROM Step_004CT_001_execute_trimming3 TO Step_005RB_001_takes_over_workpiece5  (* T_004CT_001_execute_trimming *)
  := TA_004CT_001_execute_trimming;
END_TRANSITION
STEP Step_005RB_001_takes_over_workpiece5:
  TA_005RB_001_takes_over_workpiece1(SD, T#2s);
END_STEP
TRANSITION FROM Step_005RB_001_takes_over_workpiece5 TO Step_005RB_002_positions_workpiece5  (* T_005RB_001_takes_over_workpiece1 *)
  := TA_005RB_001_takes_over_workpiece1;
END_TRANSITION
STEP Step_005RB_002_positions_workpiece5:
  TA_005RB_002_positions_workpiece1(SD, T#4s);
END_STEP
TRANSITION FROM Step_005RB_002_positions_workpiece5 TO Step_006CMM_001_execute_cmm3  (* T_005RB_002_positions_workpiece1 *)
  := TA_005RB_002_positions_workpiece1;
END_TRANSITION
STEP Step_006CMM_001_execute_cmm3:
  TA_006CMM_001_execute_cmm(SD, T#10s);
END_STEP
TRANSITION FROM Step_006CMM_001_execute_cmm3 TO (Step_010RB_100_takes_over_workpiece5, Step_007RB_001_takes_over_hinge_reinforcement3)  (* T_006CMM_001_execute_cmm *)
  := TA_006CMM_001_execute_cmm;
END_TRANSITION
STEP Step_010RB_100_takes_over_workpiece5:
  TA_010RB_100_takes_over_workpiece1(SD, T#3s);
END_STEP
TRANSITION FROM Step_010RB_100_takes_over_workpiece5 TO Step_010RB_100_positions_workpiece5  (* T_010RB_100_takes_over_workpiece1 *)
  := TA_010RB_100_TAKES_OVER_WORKPIECE1;
END_TRANSITION
STEP Step_007RB_001_takes_over_hinge_reinforcement3:
  TA_007RB_001_takes_over_hinge_reinforcement(SD, T#8s);
END_STEP
TRANSITION FROM Step_007RB_001_takes_over_hinge_reinforcement3 TO Step_007RB_002_positions_hinge_reinforcement3  (* T_007RB_001_takes_over_hinge_reinforcement *)
  := TA_007RB_001_TAKES_OVER_HINGE_REINFORCEMENT;
END_TRANSITION
STEP Step_010RB_100_positions_workpiece5:
  TA_010RB_100_positions_workpiece1(SD, T#4s);
END_STEP
STEP Step_007RB_002_positions_hinge_reinforcement3:
  TA_007RB_001_positions_hinge_reinforcement(SD, T#4s);
END_STEP
TRANSITION FROM (Step_007RB_002_positions_hinge_reinforcement3, Step_010RB_100_positions_workpiece5) TO Step_030GST100_clamps_goods3
  := TRUE;
END_TRANSITION
STEP Step_030GST100_clamps_goods3:
  TA_030GST100_clamps_goods(SD, T#1s);
END_STEP
TRANSITION FROM Step_030GST100_clamps_goods3 TO (Step_Execute_manufacturing_030RB_104, Step_Execute_manufacturing_030RB_204)  (* T_030GST100_clamps_goods *)
  := TA_030GST100_clamps_goods;
END_TRANSITION
STEP Step_Execute_manufacturing_030RB_204:
  TA_Execute_manufacturing_030RB_200(SD, T#8s);
END_STEP
TRANSITION FROM Step_Execute_manufacturing_030RB_204 TO Sys_Step_030GST100_declamps_good10  (* T_Execute_manufacturing_030RB_200 *)
  := TA_Execute_manufacturing_030RB_200;
END_TRANSITION
STEP Step_Execute_manufacturing_030RB_104:
  TA_Execute_manufacturing_030RB_100(SD, T#10s);
END_STEP
TRANSITION FROM Step_Execute_manufacturing_030RB_104 TO Sys_Step_030GST100_declamps_good9  (* T_Execute_manufacturing_030RB_100 *)
  := TA_Execute_manufacturing_030RB_100;
END_TRANSITION
STEP Sys_Step_030GST100_declamps_good9:
END_STEP
TRANSITION FROM (Sys_Step_030GST100_declamps_good9, Sys_Step_030GST100_declamps_good10) TO Step_030RB_300_takes_over_good3
  := TRUE;
END_TRANSITION
STEP Sys_Step_030GST100_declamps_good10:
END_STEP
STEP Step_030RB_300_takes_over_good3:
  TA_030RB_300_takes_over_good(SD, T#3s);
END_STEP
TRANSITION FROM Step_030RB_300_takes_over_good3 TO Step_030RB_300_positions_good3  (* T_030RB_300_takes_over_good *)
  := TA_030RB_300_takes_over_good;
END_TRANSITION
STEP Step_030RB_300_positions_good3:
  TA_030RB_300_positions_good(SD, T#4s);
END_STEP
TRANSITION FROM Step_030RB_300_positions_good3 TO Step_010UT_001_execute_inspection3  (* T_030RB_300_positions_good *)
  := TA_030RB_300_POSITIONS_GOOD;
END_TRANSITION
STEP Step_010UT_001_execute_inspection3:
  TA_010UT_001_execute_inspection(SD, T#10s);
END_STEP
TRANSITION FROM Step_010UT_001_execute_inspection3 TO Step_001RB_001_takes_over_blank4  (* T_010UT_001_execute_inspection *)
  := TA_010UT_001_execute_inspection;
END_TRANSITION
STEP Step_001RB_001_takes_over_blank4:
  TA_RESET(P);
  TA_010RB_100_takes_over_workpiece1(R);
  TA_010RB_100_positions_workpiece1(R);
  TA_030GST100_clamps_goods(R);
  TA_Execute_manufacturing_030RB_100(R);
  TA_Execute_manufacturing_030RB_200(R);
  TA_030GST100_declamps_good(R);
  TA_030RB_300_takes_over_good(R);
  TA_001RB_001_takes_over_blank(R);
  TA_001RB_002_positions_blank(R);
  TA_002DDP_001_execute_forming(R);
  TA_003RB_001_takes_over_workpiece1(R);
  TA_003RB_002_positions_workpiece1(R);
  TA_004CT_001_execute_trimming(R);
  TA_005RB_001_takes_over_workpiece1(R);
  TA_005RB_002_positions_workpiece1(R);
  TA_006CMM_001_execute_cmm(R);
  TA_007RB_001_takes_over_hinge_reinforcement(R);
  TA_007RB_001_positions_hinge_reinforcement(R);
  TA_030RB_300_positions_good(R);
  TA_010UT_001_execute_inspection(R);
END_STEP
TRANSITION FROM Step_001RB_001_takes_over_blank4 TO Step_001RB_002_positions_blank4
  := TRUE;
END_TRANSITION
STEP Step_001RB_002_positions_blank4:
  TA_001RB_002_positions_blank(SD, T#2s);
END_STEP
TRANSITION FROM Step_001RB_002_positions_blank4 TO Step_002DDP_001_execute_forming4  (* T_001RB_002_positions_blank *)
  := TA_001RB_002_positions_blank;
END_TRANSITION
STEP Step_002DDP_001_execute_forming4:
  TA_002DDP_001_execute_forming(SD, T#6s);
END_STEP
TRANSITION FROM Step_002DDP_001_execute_forming4 TO Step_003RB_001_takes_over_workpiece6  (* T_002DDP_001_execute_forming *)
  := TA_002DDP_001_EXECUTE_FORMING;
END_TRANSITION
STEP Step_003RB_001_takes_over_workpiece6:
  TA_003RB_001_takes_over_workpiece1(SD, T#4s);
END_STEP
TRANSITION FROM Step_003RB_001_takes_over_workpiece6 TO Step_003RB_002_positions_workpiece6  (* T_003RB_001_takes_over_workpiece1 *)
  := TA_003RB_001_takes_over_workpiece1;
END_TRANSITION
STEP Step_003RB_002_positions_workpiece6:
  TA_003RB_002_positions_workpiece1(SD, T#2s);
END_STEP
TRANSITION FROM Step_003RB_002_positions_workpiece6 TO Step_004CT_001_execute_trimming4  (* T_003RB_002_positions_workpiece1 *)
  := TA_003RB_002_positions_workpiece1;
END_TRANSITION
STEP Step_004CT_001_execute_trimming4:
  TA_004CT_001_execute_trimming(SD, T#3s);
END_STEP
TRANSITION FROM Step_004CT_001_execute_trimming4 TO Step_005RB_001_takes_over_workpiece6  (* T_004CT_001_execute_trimming *)
  := TA_004CT_001_execute_trimming;
END_TRANSITION
STEP Step_005RB_001_takes_over_workpiece6:
  TA_005RB_001_takes_over_workpiece1(SD, T#2s);
END_STEP
TRANSITION FROM Step_005RB_001_takes_over_workpiece6 TO Step_005RB_002_positions_workpiece6  (* T_005RB_001_takes_over_workpiece1 *)
  := TA_005RB_001_takes_over_workpiece1;
END_TRANSITION
STEP Step_005RB_002_positions_workpiece6:
  TA_005RB_002_positions_workpiece1(SD, T#4s);
END_STEP
TRANSITION FROM Step_005RB_002_positions_workpiece6 TO Step_006CMM_001_execute_cmm4  (* T_005RB_002_positions_workpiece1 *)
  := TA_005RB_002_positions_workpiece1;
END_TRANSITION
STEP Step_006CMM_001_execute_cmm4:
  TA_006CMM_001_execute_cmm(SD, T#10s);
END_STEP
TRANSITION FROM Step_006CMM_001_execute_cmm4 TO (Step_010RB_100_takes_over_workpiece6, Step_007RB_001_takes_over_hinge_reinforcement4)  (* T_006CMM_001_execute_cmm *)
  := TA_006CMM_001_execute_cmm;
END_TRANSITION
STEP Step_010RB_100_takes_over_workpiece6:
  TA_010RB_100_takes_over_workpiece1(SD, T#3s);
END_STEP
TRANSITION FROM Step_010RB_100_takes_over_workpiece6 TO Step_010RB_100_positions_workpiece6  (* T_010RB_100_takes_over_workpiece1 *)
  := TA_010RB_100_TAKES_OVER_WORKPIECE1;
END_TRANSITION
STEP Step_007RB_001_takes_over_hinge_reinforcement4:
  TA_007RB_001_takes_over_hinge_reinforcement(SD, T#8s);
END_STEP
TRANSITION FROM Step_007RB_001_takes_over_hinge_reinforcement4 TO Step_007RB_002_positions_hinge_reinforcement4  (* T_007RB_001_takes_over_hinge_reinforcement *)
  := TA_007RB_001_TAKES_OVER_HINGE_REINFORCEMENT;
END_TRANSITION
STEP Step_010RB_100_positions_workpiece6:
  TA_010RB_100_positions_workpiece1(SD, T#4s);
END_STEP
STEP Step_007RB_002_positions_hinge_reinforcement4:
  TA_007RB_001_positions_hinge_reinforcement(SD, T#4s);
END_STEP
TRANSITION FROM (Step_007RB_002_positions_hinge_reinforcement4, Step_010RB_100_positions_workpiece6) TO Step_030GST100_clamps_goods4
  := TRUE;
END_TRANSITION
STEP Step_030GST100_clamps_goods4:
  TA_030GST100_clamps_goods(SD, T#1s);
END_STEP
TRANSITION FROM Step_030GST100_clamps_goods4 TO (Step_Execute_manufacturing_030RB_105, Step_Execute_manufacturing_030RB_205)  (* T_030GST100_clamps_goods *)
  := TA_030GST100_clamps_goods;
END_TRANSITION
STEP Step_Execute_manufacturing_030RB_205:
  TA_Execute_manufacturing_030RB_200(SD, T#8s);
END_STEP
TRANSITION FROM Step_Execute_manufacturing_030RB_205 TO Sys_Step_030GST100_declamps_good12  (* T_Execute_manufacturing_030RB_200 *)
  := TA_Execute_manufacturing_030RB_200;
END_TRANSITION
STEP Step_Execute_manufacturing_030RB_105:
  TA_Execute_manufacturing_030RB_100(SD, T#10s);
END_STEP
TRANSITION FROM Step_Execute_manufacturing_030RB_105 TO Sys_Step_030GST100_declamps_good11  (* T_Execute_manufacturing_030RB_100 *)
  := TA_Execute_manufacturing_030RB_100;
END_TRANSITION
STEP Sys_Step_030GST100_declamps_good11:
END_STEP
TRANSITION FROM (Sys_Step_030GST100_declamps_good11, Sys_Step_030GST100_declamps_good12) TO Step_030RB_300_takes_over_good4
  := TRUE;
END_TRANSITION
STEP Sys_Step_030GST100_declamps_good12:
END_STEP
STEP Step_030RB_300_takes_over_good4:
  TA_030RB_300_takes_over_good(SD, T#3s);
END_STEP
TRANSITION FROM Step_030RB_300_takes_over_good4 TO Step_030RB_300_positions_good4  (* T_030RB_300_takes_over_good *)
  := TA_030RB_300_takes_over_good;
END_TRANSITION
STEP Step_030RB_300_positions_good4:
  TA_030RB_300_positions_good(SD, T#4s);
END_STEP
TRANSITION FROM Step_030RB_300_positions_good4 TO Step_010UT_001_execute_inspection4  (* T_030RB_300_positions_good *)
  := TA_030RB_300_POSITIONS_GOOD;
END_TRANSITION
STEP Step_010UT_001_execute_inspection4:
  TA_010UT_001_execute_inspection(SD, T#10s);
END_STEP
TRANSITION FROM Step_010UT_001_execute_inspection4 TO Step_001RB_001_takes_over_blank5  (* T_010UT_001_execute_inspection *)
  := TA_010UT_001_execute_inspection;
END_TRANSITION
STEP Step_001RB_001_takes_over_blank5:
  TA_RESET(P);
  TA_010RB_100_takes_over_workpiece1(R);
  TA_010RB_100_positions_workpiece1(R);
  TA_030GST100_clamps_goods(R);
  TA_Execute_manufacturing_030RB_100(R);
  TA_Execute_manufacturing_030RB_200(R);
  TA_030GST100_declamps_good(R);
  TA_030RB_300_takes_over_good(R);
  TA_001RB_001_takes_over_blank(R);
  TA_001RB_002_positions_blank(R);
  TA_002DDP_001_execute_forming(R);
  TA_003RB_001_takes_over_workpiece1(R);
  TA_003RB_002_positions_workpiece1(R);
  TA_004CT_001_execute_trimming(R);
  TA_005RB_001_takes_over_workpiece1(R);
  TA_005RB_002_positions_workpiece1(R);
  TA_006CMM_001_execute_cmm(R);
  TA_007RB_001_takes_over_hinge_reinforcement(R);
  TA_007RB_001_positions_hinge_reinforcement(R);
  TA_030RB_300_positions_good(R);
  TA_010UT_001_execute_inspection(R);
END_STEP
TRANSITION FROM Step_001RB_001_takes_over_blank5 TO Step_001RB_002_positions_blank5
  := TRUE;
END_TRANSITION
STEP Step_001RB_002_positions_blank5:
  TA_001RB_002_positions_blank(SD, T#2s);
END_STEP
TRANSITION FROM Step_001RB_002_positions_blank5 TO Step_002DDP_001_execute_forming5  (* T_001RB_002_positions_blank *)
  := TA_001RB_002_positions_blank;
END_TRANSITION
STEP Step_002DDP_001_execute_forming5:
  TA_002DDP_001_execute_forming(SD, T#6s);
END_STEP
TRANSITION FROM Step_002DDP_001_execute_forming5 TO Step_003RB_001_takes_over_workpiece7  (* T_002DDP_001_execute_forming *)
  := TA_002DDP_001_EXECUTE_FORMING;
END_TRANSITION
STEP Step_003RB_001_takes_over_workpiece7:
  TA_003RB_001_takes_over_workpiece1(SD, T#4s);
END_STEP
TRANSITION FROM Step_003RB_001_takes_over_workpiece7 TO Step_003RB_002_positions_workpiece7  (* T_003RB_001_takes_over_workpiece1 *)
  := TA_003RB_001_takes_over_workpiece1;
END_TRANSITION
STEP Step_003RB_002_positions_workpiece7:
  TA_003RB_002_positions_workpiece1(SD, T#2s);
END_STEP
TRANSITION FROM Step_003RB_002_positions_workpiece7 TO Step_004CT_001_execute_trimming5  (* T_003RB_002_positions_workpiece1 *)
  := TA_003RB_002_positions_workpiece1;
END_TRANSITION
STEP Step_004CT_001_execute_trimming5:
  TA_004CT_001_execute_trimming(SD, T#3s);
END_STEP
TRANSITION FROM Step_004CT_001_execute_trimming5 TO Step_005RB_001_takes_over_workpiece7  (* T_004CT_001_execute_trimming *)
  := TA_004CT_001_execute_trimming;
END_TRANSITION
STEP Step_005RB_001_takes_over_workpiece7:
  TA_005RB_001_takes_over_workpiece1(SD, T#2s);
END_STEP
TRANSITION FROM Step_005RB_001_takes_over_workpiece7 TO Step_005RB_002_positions_workpiece7  (* T_005RB_001_takes_over_workpiece1 *)
  := TA_005RB_001_takes_over_workpiece1;
END_TRANSITION
STEP Step_005RB_002_positions_workpiece7:
  TA_005RB_002_positions_workpiece1(SD, T#4s);
END_STEP
TRANSITION FROM Step_005RB_002_positions_workpiece7 TO Step_006CMM_001_execute_cmm5  (* T_005RB_002_positions_workpiece1 *)
  := TA_005RB_002_positions_workpiece1;
END_TRANSITION
STEP Step_006CMM_001_execute_cmm5:
  TA_006CMM_001_execute_cmm(SD, T#10s);
END_STEP
TRANSITION FROM Step_006CMM_001_execute_cmm5 TO (Step_010RB_100_takes_over_workpiece7, Step_007RB_001_takes_over_hinge_reinforcement5)  (* T_006CMM_001_execute_cmm *)
  := TA_006CMM_001_execute_cmm;
END_TRANSITION
STEP Step_010RB_100_takes_over_workpiece7:
  TA_010RB_100_takes_over_workpiece1(SD, T#3s);
END_STEP
TRANSITION FROM Step_010RB_100_takes_over_workpiece7 TO Step_010RB_100_positions_workpiece7  (* T_010RB_100_takes_over_workpiece1 *)
  := TA_010RB_100_TAKES_OVER_WORKPIECE1;
END_TRANSITION
STEP Step_007RB_001_takes_over_hinge_reinforcement5:
  TA_007RB_001_takes_over_hinge_reinforcement(SD, T#8s);
END_STEP
TRANSITION FROM Step_007RB_001_takes_over_hinge_reinforcement5 TO Step_007RB_002_positions_hinge_reinforcement5  (* T_007RB_001_takes_over_hinge_reinforcement *)
  := TA_007RB_001_TAKES_OVER_HINGE_REINFORCEMENT;
END_TRANSITION
STEP Step_010RB_100_positions_workpiece7:
  TA_010RB_100_positions_workpiece1(SD, T#4s);
END_STEP
STEP Step_007RB_002_positions_hinge_reinforcement5:
  TA_007RB_001_positions_hinge_reinforcement(SD, T#4s);
END_STEP
TRANSITION FROM (Step_007RB_002_positions_hinge_reinforcement5, Step_010RB_100_positions_workpiece7) TO Step_030GST100_clamps_goods5
  := TRUE;
END_TRANSITION
STEP Step_030GST100_clamps_goods5:
  TA_030GST100_clamps_goods(SD, T#1s);
END_STEP
TRANSITION FROM Step_030GST100_clamps_goods5 TO (Step_Execute_manufacturing_030RB_106, Step_Execute_manufacturing_030RB_206)  (* T_030GST100_clamps_goods *)
  := TA_030GST100_clamps_goods;
END_TRANSITION
STEP Step_Execute_manufacturing_030RB_206:
  TA_Execute_manufacturing_030RB_200(SD, T#8s);
END_STEP
TRANSITION FROM Step_Execute_manufacturing_030RB_206 TO Sys_Step_030GST100_declamps_good14  (* T_Execute_manufacturing_030RB_200 *)
  := TA_Execute_manufacturing_030RB_200;
END_TRANSITION
STEP Step_Execute_manufacturing_030RB_106:
  TA_Execute_manufacturing_030RB_100(SD, T#10s);
END_STEP
TRANSITION FROM Step_Execute_manufacturing_030RB_106 TO Sys_Step_030GST100_declamps_good13  (* T_Execute_manufacturing_030RB_100 *)
  := TA_Execute_manufacturing_030RB_100;
END_TRANSITION
STEP Sys_Step_030GST100_declamps_good13:
END_STEP
TRANSITION FROM (Sys_Step_030GST100_declamps_good13, Sys_Step_030GST100_declamps_good14) TO Step_030RB_300_takes_over_good5
  := TRUE;
END_TRANSITION
STEP Sys_Step_030GST100_declamps_good14:
END_STEP
STEP Step_030RB_300_takes_over_good5:
  TA_030RB_300_takes_over_good(SD, T#3s);
END_STEP
TRANSITION FROM Step_030RB_300_takes_over_good5 TO Step_030RB_300_positions_good5  (* T_030RB_300_takes_over_good *)
  := TA_030RB_300_takes_over_good;
END_TRANSITION
STEP Step_030RB_300_positions_good5:
  TA_030RB_300_positions_good(SD, T#4s);
END_STEP
TRANSITION FROM Step_030RB_300_positions_good5 TO Step_010UT_001_execute_inspection5  (* T_030RB_300_positions_good *)
  := TA_030RB_300_POSITIONS_GOOD;
END_TRANSITION
STEP Step_010UT_001_execute_inspection5:
  TA_010UT_001_execute_inspection(SD, T#10s);
END_STEP
TRANSITION FROM Step_010UT_001_execute_inspection5 TO Step_001RB_001_takes_over_blank6  (* T_010UT_001_execute_inspection *)
  := TA_010UT_001_execute_inspection;
END_TRANSITION
STEP Step_001RB_001_takes_over_blank6:
  TA_RESET(P);
  TA_010RB_100_takes_over_workpiece1(R);
  TA_010RB_100_positions_workpiece1(R);
  TA_030GST100_clamps_goods(R);
  TA_Execute_manufacturing_030RB_100(R);
  TA_Execute_manufacturing_030RB_200(R);
  TA_030GST100_declamps_good(R);
  TA_030RB_300_takes_over_good(R);
  TA_001RB_001_takes_over_blank(R);
  TA_001RB_002_positions_blank(R);
  TA_002DDP_001_execute_forming(R);
  TA_003RB_001_takes_over_workpiece1(R);
  TA_003RB_002_positions_workpiece1(R);
  TA_004CT_001_execute_trimming(R);
  TA_005RB_001_takes_over_workpiece1(R);
  TA_005RB_002_positions_workpiece1(R);
  TA_006CMM_001_execute_cmm(R);
  TA_007RB_001_takes_over_hinge_reinforcement(R);
  TA_007RB_001_positions_hinge_reinforcement(R);
  TA_030RB_300_positions_good(R);
  TA_010UT_001_execute_inspection(R);
END_STEP
TRANSITION FROM Step_001RB_001_takes_over_blank6 TO Step_001RB_002_positions_blank6
  := TRUE;
END_TRANSITION
STEP Step_001RB_002_positions_blank6:
  TA_001RB_002_positions_blank(SD, T#2s);
END_STEP
TRANSITION FROM Step_001RB_002_positions_blank6 TO Step_002DDP_001_execute_forming6  (* T_001RB_002_positions_blank *)
  := TA_001RB_002_positions_blank;
END_TRANSITION
STEP Step_002DDP_001_execute_forming6:
  TA_002DDP_001_execute_forming(SD, T#6s);
END_STEP
TRANSITION FROM Step_002DDP_001_execute_forming6 TO Step_003RB_001_takes_over_workpiece8  (* T_002DDP_001_execute_forming *)
  := TA_002DDP_001_EXECUTE_FORMING;
END_TRANSITION
STEP Step_003RB_001_takes_over_workpiece8:
  TA_003RB_001_takes_over_workpiece1(SD, T#4s);
END_STEP
TRANSITION FROM Step_003RB_001_takes_over_workpiece8 TO Step_003RB_002_positions_workpiece8  (* T_003RB_001_takes_over_workpiece1 *)
  := TA_003RB_001_takes_over_workpiece1;
END_TRANSITION
STEP Step_003RB_002_positions_workpiece8:
  TA_003RB_002_positions_workpiece1(SD, T#2s);
END_STEP
TRANSITION FROM Step_003RB_002_positions_workpiece8 TO Step_004CT_001_execute_trimming6  (* T_003RB_002_positions_workpiece1 *)
  := TA_003RB_002_positions_workpiece1;
END_TRANSITION
STEP Step_004CT_001_execute_trimming6:
  TA_004CT_001_execute_trimming(SD, T#3s);
END_STEP
TRANSITION FROM Step_004CT_001_execute_trimming6 TO Step_005RB_001_takes_over_workpiece8  (* T_004CT_001_execute_trimming *)
  := TA_004CT_001_execute_trimming;
END_TRANSITION
STEP Step_005RB_001_takes_over_workpiece8:
  TA_005RB_001_takes_over_workpiece1(SD, T#2s);
END_STEP
TRANSITION FROM Step_005RB_001_takes_over_workpiece8 TO Step_005RB_002_positions_workpiece8  (* T_005RB_001_takes_over_workpiece1 *)
  := TA_005RB_001_takes_over_workpiece1;
END_TRANSITION
STEP Step_005RB_002_positions_workpiece8:
  TA_005RB_002_positions_workpiece1(SD, T#4s);
END_STEP
TRANSITION FROM Step_005RB_002_positions_workpiece8 TO Step_006CMM_001_execute_cmm6  (* T_005RB_002_positions_workpiece1 *)
  := TA_005RB_002_positions_workpiece1;
END_TRANSITION
STEP Step_006CMM_001_execute_cmm6:
  TA_006CMM_001_execute_cmm(SD, T#10s);
END_STEP
TRANSITION FROM Step_006CMM_001_execute_cmm6 TO (Step_010RB_100_takes_over_workpiece8, Step_007RB_001_takes_over_hinge_reinforcement6)  (* T_006CMM_001_execute_cmm *)
  := TA_006CMM_001_execute_cmm;
END_TRANSITION
STEP Step_010RB_100_takes_over_workpiece8:
  TA_010RB_100_takes_over_workpiece1(SD, T#3s);
END_STEP
TRANSITION FROM Step_010RB_100_takes_over_workpiece8 TO Step_010RB_100_positions_workpiece8  (* T_010RB_100_takes_over_workpiece1 *)
  := TA_010RB_100_TAKES_OVER_WORKPIECE1;
END_TRANSITION
STEP Step_007RB_001_takes_over_hinge_reinforcement6:
  TA_007RB_001_takes_over_hinge_reinforcement(SD, T#8s);
END_STEP
TRANSITION FROM Step_007RB_001_takes_over_hinge_reinforcement6 TO Step_007RB_002_positions_hinge_reinforcement6  (* T_007RB_001_takes_over_hinge_reinforcement *)
  := TA_007RB_001_TAKES_OVER_HINGE_REINFORCEMENT;
END_TRANSITION
STEP Step_010RB_100_positions_workpiece8:
  TA_010RB_100_positions_workpiece1(SD, T#4s);
END_STEP
STEP Step_007RB_002_positions_hinge_reinforcement6:
  TA_007RB_001_positions_hinge_reinforcement(SD, T#4s);
END_STEP
TRANSITION FROM (Step_007RB_002_positions_hinge_reinforcement6, Step_010RB_100_positions_workpiece8) TO Step_030GST100_clamps_goods6
  := TRUE;
END_TRANSITION
STEP Step_030GST100_clamps_goods6:
  TA_030GST100_clamps_goods(SD, T#1s);
END_STEP
TRANSITION FROM Step_030GST100_clamps_goods6 TO (Step_Execute_manufacturing_030RB_107, Step_Execute_manufacturing_030RB_207)  (* T_030GST100_clamps_goods *)
  := TA_030GST100_clamps_goods;
END_TRANSITION
STEP Step_Execute_manufacturing_030RB_207:
  TA_Execute_manufacturing_030RB_200(SD, T#8s);
END_STEP
TRANSITION FROM Step_Execute_manufacturing_030RB_207 TO Sys_Step_030GST100_declamps_good16  (* T_Execute_manufacturing_030RB_200 *)
  := TA_Execute_manufacturing_030RB_200;
END_TRANSITION
STEP Step_Execute_manufacturing_030RB_107:
  TA_Execute_manufacturing_030RB_100(SD, T#10s);
END_STEP
TRANSITION FROM Step_Execute_manufacturing_030RB_107 TO Sys_Step_030GST100_declamps_good15  (* T_Execute_manufacturing_030RB_100 *)
  := TA_Execute_manufacturing_030RB_100;
END_TRANSITION
STEP Sys_Step_030GST100_declamps_good15:
END_STEP
TRANSITION FROM (Sys_Step_030GST100_declamps_good15, Sys_Step_030GST100_declamps_good16) TO Step_030RB_300_takes_over_good6
  := TRUE;
END_TRANSITION
STEP Sys_Step_030GST100_declamps_good16:
END_STEP
STEP Step_030RB_300_takes_over_good6:
  TA_030RB_300_takes_over_good(SD, T#3s);
END_STEP
TRANSITION FROM Step_030RB_300_takes_over_good6 TO Step_030RB_300_positions_good6  (* T_030RB_300_takes_over_good *)
  := TA_030RB_300_takes_over_good;
END_TRANSITION
STEP Step_030RB_300_positions_good6:
  TA_030RB_300_positions_good(SD, T#4s);
END_STEP
TRANSITION FROM Step_030RB_300_positions_good6 TO Step_010UT_001_execute_inspection6  (* T_030RB_300_positions_good *)
  := TA_030RB_300_POSITIONS_GOOD;
END_TRANSITION
STEP Step_010UT_001_execute_inspection6:
  TA_010UT_001_execute_inspection(SD, T#10s);
END_STEP
TRANSITION FROM Step_010UT_001_execute_inspection6 TO TerminalStep  (* T_010UT_001_execute_inspection *)
  := TA_010UT_001_execute_inspection;
END_TRANSITION
STEP TerminalStep:
  TA_RESET(P);
  TA_010RB_100_takes_over_workpiece1(R);
  TA_010RB_100_positions_workpiece1(R);
  TA_030GST100_clamps_goods(R);
  TA_Execute_manufacturing_030RB_100(R);
  TA_Execute_manufacturing_030RB_200(R);
  TA_030GST100_declamps_good(R);
  TA_030RB_300_takes_over_good(R);
  TA_001RB_001_takes_over_blank(R);
  TA_001RB_002_positions_blank(R);
  TA_002DDP_001_execute_forming(R);
  TA_003RB_001_takes_over_workpiece1(R);
  TA_003RB_002_positions_workpiece1(R);
  TA_004CT_001_execute_trimming(R);
  TA_005RB_001_takes_over_workpiece1(R);
  TA_005RB_002_positions_workpiece1(R);
  TA_006CMM_001_execute_cmm(R);
  TA_007RB_001_takes_over_hinge_reinforcement(R);
  TA_007RB_001_positions_hinge_reinforcement(R);
  TA_030RB_300_positions_good(R);
  TA_010UT_001_execute_inspection(R);
END_STEP
TRANSITION FROM TerminalStep TO InitialStep_ActivityOnNodeNetwork
  := TRUE;
END_TRANSITION

ACTION DA_010RB_100_takes_over_workpiece1:
                
              
END_ACTION

ACTION TA_010RB_100_takes_over_workpiece1:
                TA_010RB_100_takes_over_workpiece1 := TRUE;
              
END_ACTION

ACTION DA_010RB_100_positions_goods:
                
              
END_ACTION

ACTION TA_010RB_100_positions_workpiece1:
                TA_010RB_100_positions_workpiece1 := TRUE;
              
END_ACTION

ACTION DA_030GST100_clamps_goods:
                
              
END_ACTION

ACTION TA_030GST100_clamps_goods:
                TA_030GST100_clamps_goods := TRUE;
              
END_ACTION

ACTION DA_Execute_manufacturing_030RB_100:
                
              
END_ACTION

ACTION TA_Execute_manufacturing_030RB_100:
                TA_EXECUTE_MANUFACTURING_030RB_100 := TRUE;
              
END_ACTION

ACTION DA_Execute_manufacturing_030RB_200:
                
              
END_ACTION

ACTION TA_Execute_manufacturing_030RB_200:
                TA_EXECUTE_MANUFACTURING_030RB_200 := TRUE;
              
END_ACTION

ACTION DA_030GST100_declamps_good:
                
              
END_ACTION

ACTION TA_030GST100_declamps_good:
                TA_030GST100_DECLAMPS_GOOD := TRUE;
              
END_ACTION

ACTION DA_030RB_300_takes_over_good:
                
              
END_ACTION

ACTION TA_030RB_300_takes_over_good:
                TA_030RB_300_TAKES_OVER_GOOD := TRUE;
              
END_ACTION

ACTION TA_RESET:
                TA_010RB_100_takes_over_workpiece1 := FALSE;
TA_010RB_100_positions_workpiece1 := FALSE;
TA_EXECUTE_MANUFACTURING_030RB_100 := FALSE;
TA_EXECUTE_MANUFACTURING_030RB_200 := FALSE;
TA_030GST100_clamps_goods := FALSE;
TA_030GST100_DECLAMPS_GOOD := FALSE;
TA_030RB_300_TAKES_OVER_GOOD := FALSE;
              
END_ACTION

ACTION TA_001RB_001_takes_over_blank:
                TA_001RB_001_takes_over_blank := TRUE;
              
END_ACTION

ACTION TA_001RB_002_positions_blank:
                TA_001RB_002_positions_blank := TRUE;
              
END_ACTION

ACTION TA_002DDP_001_execute_forming:
                TA_002DDP_001_execute_forming := TRUE;

              
END_ACTION

ACTION TA_003RB_001_takes_over_workpiece1:
                TA_003RB_001_takes_over_workpiece1 := TRUE;
              
END_ACTION

ACTION TA_003RB_002_positions_workpiece1:
                TA_003RB_002_positions_workpiece1 := TRUE;
              
END_ACTION

ACTION TA_004CT_001_execute_trimming:
                TA_004CT_001_EXECUTE_TRIMMING := TRUE;
              
END_ACTION

ACTION TA_005RB_001_takes_over_workpiece1:
                TA_005RB_001_takes_over_workpiece1 := TRUE;
              
END_ACTION

ACTION TA_005RB_002_positions_workpiece1:
                TA_005RB_002_positions_workpiece1 := TRUE;
              
END_ACTION

ACTION TA_006CMM_001_execute_cmm:
                TA_006CMM_001_execute_cmm := TRUE;
              
END_ACTION

ACTION TA_007RB_001_takes_over_hinge_reinforcement:
                TA_007RB_001_TAKES_OVER_HINGE_REINFORCEMENT := TRUE;
              
END_ACTION

ACTION TA_007RB_001_positions_hinge_reinforcement:
                TA_007RB_001_POSITIONS_HINGE_REINFORCEMENT := TRUE;
              
END_ACTION

ACTION TA_030RB_300_positions_good:
                TA_030RB_300_positions_good := TRUE;
              
END_ACTION

ACTION TA_010UT_001_execute_inspection:
                TA_010UT_001_execute_inspection := TRUE;
              
END_ACTION
END_PROGRAM

CONFIGURATION Config0
  RESOURCE Res0 ON PLC
    TASK task0(INTERVAL := T#20ms, PRIORITY := 0);
    PROGRAM instance0 WITH task0 : Sequencing_Station_ActivityOnNodeNetwork;
  END_RESOURCE
END_CONFIGURATION
